LIN {X 0,Y 361.876,Z 72.401,A -85,B 0,C 180,E1 -13014.655,E2 -13014.655} C_VEL
LIN {X 0,Y 361.897,Z 72.531,A -85,B 0,C 180,E1 -13018.09,E2 -13018.09} C_VEL
LIN {X 0,Y 364.94,Z 85.338,A -85,B 0,C 180,E1 -13021.503,E2 -13021.503} C_VEL
LIN {X 0,Y 366.727,Z 94.642,A -85,B 0,C 180,E1 -13023.846,E2 -13023.846} C_VEL
LIN {X 0,Y 366.002,Z 102.488,A -85,B 0,C 180,E1 -13025.616,E2 -13025.616} C_VEL
LIN {X 0,Y 365.33,Z 108.755,A -85,B 0,C 180,E1 -13027.012,E2 -13027.012} C_VEL
LIN {X 0,Y 370.356,Z 135.443,A -85,B 0,C 180,E1 -13027.952,E2 -13027.952} C_VEL
LIN {X 0,Y 371.965,Z 146.662,A -85,B 0,C 180,E1 -13028.297,E2 -13028.297} C_VEL
LIN {X 0,Y 370.571,Z 218.065,A -85,B 0,C 180,E1 -13029.713,E2 -13029.713} C_VEL
LIN {X 0,Y 369.771,Z 231.878,A -85,B 0,C 180,E1 -13030.211,E2 -13030.211} C_VEL
LIN {X 0,Y 368.776,Z 244.274,A -85,B 0,C 180,E1 -13030.879,E2 -13030.879} C_VEL
LIN {X 0,Y 367.552,Z 256.145,A -85,B 0,C 180,E1 -13031.753,E2 -13031.753} C_VEL
LIN {X 0,Y 366.174,Z 267.553,A -85,B 0,C 180,E1 -13032.836,E2 -13032.836} C_VEL
LIN {X 0,Y 364.919,Z 277.858,A -85,B 0,C 180,E1 -13034.071,E2 -13034.071} C_VEL
LIN {X 0,Y 363.726,Z 287.134,A -85,B 0,C 180,E1 -13035.452,E2 -13035.452} C_VEL
LIN {X 0,Y 362.602,Z 296.152,A -85,B 0,C 180,E1 -13037.121,E2 -13037.121} C_VEL
LIN {X 0,Y 361.604,Z 303.436,A -85,B 0,C 180,E1 -13038.793,E2 -13038.793} C_VEL
LIN {X 0,Y 360.994,Z 309.293,A -85,B 0,C 180,E1 -13040.474,E2 -13040.474} C_VEL
LIN {X 0,Y 360.61,Z 313.923,A -85,B 0,C 180,E1 -13042.159,E2 -13042.159} C_VEL
LIN {X 0,Y 360.423,Z 317.693,A -85,B 0,C 180,E1 -13043.97,E2 -13043.97} C_VEL
LIN {X 0,Y 360.359,Z 320.002,A -85,B 0,C 180,E1 -13045.525,E2 -13045.525} C_VEL
LIN {X 0,Y 360.323,Z 321.192,A -85,B 0,C 180,E1 -13046.645,E2 -13046.645} C_VEL
LIN {X 0,Y 360.456,Z 322.312,A -85,B 0,C 180,E1 -13048.882,E2 -13048.882} C_VEL
LIN {X 0,Y 360.483,Z 322.289,A -85,B 0,C 180,E1 -13050,E2 -13050} C_VEL
LIN {X 0,Y 360.462,Z 321.871,A -85,B 0,C 180,E1 -13051.117,E2 -13051.117} C_VEL
LIN {X 0,Y 360.398,Z 321.01,A -85,B 0,C 180,E1 -13052.235,E2 -13052.235} C_VEL
LIN {X 0,Y 360.419,Z 318.073,A -85,B 0,C 180,E1 -13054.473,E2 -13054.473} C_VEL
LIN {X 0,Y 360.357,Z 314.691,A -85,B 0,C 180,E1 -13056.157,E2 -13056.157} C_VEL
LIN {X 0,Y 360.594,Z 310.228,A -85,B 0,C 180,E1 -13057.841,E2 -13057.841} C_VEL
LIN {X 0,Y 360.902,Z 304.546,A -85,B 0,C 180,E1 -13059.527,E2 -13059.527} C_VEL
LIN {X 0,Y 361.389,Z 297.422,A -85,B 0,C 180,E1 -13061.214,E2 -13061.214} C_VEL
LIN {X 0,Y 362.224,Z 288.522,A -85,B 0,C 180,E1 -13062.892,E2 -13062.892} C_VEL
LIN {X 0,Y 363.1,Z 279.397,A -85,B 0,C 180,E1 -13064.287,E2 -13064.287} C_VEL
LIN {X 0,Y 363.801,Z 269.428,A -85,B 0,C 180,E1 -13065.533,E2 -13065.533} C_VEL
LIN {X 0,Y 364.89,Z 258.101,A -85,B 0,C 180,E1 -13066.648,E2 -13066.648} C_VEL
LIN {X 0,Y 365.851,Z 245.515,A -85,B 0,C 180,E1 -13067.611,E2 -13067.611} C_VEL
LIN {X 0,Y 366.722,Z 232.662,A -85,B 0,C 180,E1 -13068.325,E2 -13068.325} C_VEL
LIN {X 0,Y 367.337,Z 218.902,A -85,B 0,C 180,E1 -13068.835,E2 -13068.835} C_VEL
LIN {X 0,Y 368.208,Z 162.822,A -85,B 0,C 180,E1 -13069.954,E2 -13069.954} C_VEL
LIN {X 0,Y 368.392,Z 143.971,A -85,B 0,C 180,E1 -13070.322,E2 -13070.322} C_VEL
LIN {X 0,Y 363.707,Z 109.248,A -85,B 0,C 180,E1 -13071.263,E2 -13071.263} C_VEL
LIN {X 0,Y 365.256,Z 90.835,A -85,B 0,C 180,E1 -13075.265,E2 -13075.265} C_VEL
LIN {X 0,Y 364.505,Z 85.088,A -85,B 0,C 180,E1 -13076.6,E2 -13076.6} C_VEL
LIN {X 0,Y 361.928,Z 72.512,A -85,B 0,C 180,E1 -13079.648,E2 -13079.648} C_VEL
LIN {X 0,Y 361.86,Z 72.408,A -85,B 0,C 180,E1 -13083.369,E2 -13083.369} C_VEL
LIN {X 0,Y 361.873,Z 72.406,A -85,B 0,C 180,E1 -13087.017,E2 -13087.017} C_VEL
LIN {X 0,Y 361.856,Z 72.412,A -85,B 0,C 180,E1 -13089.861,E2 -13089.861} C_VEL
LIN {X 0,Y 361.836,Z 72.41,A -85,B 0,C 180,E1 -13092.829,E2 -13092.829} C_VEL
LIN {X 0,Y 361.817,Z 72.414,A -85,B 0,C 180,E1 -13095.946,E2 -13095.946} C_VEL
LIN {X 0,Y 361.835,Z 72.415,A -85,B 0,C 180,E1 -13099.244,E2 -13099.244} C_VEL
LIN {X 0,Y 361.862,Z 72.408,A -85,B 0,C 180,E1 -13102.777,E2 -13102.777} C_VEL
LIN {X 0,Y 361.853,Z 72.409,A -85,B 0,C 180,E1 -13105.72,E2 -13105.72} C_VEL
LIN {X 0,Y 361.874,Z 72.406,A -85,B 0,C 180,E1 -13109.672,E2 -13109.672} C_VEL
LIN {X 0,Y 361.953,Z 72.397,A -85,B 0,C 180,E1 -13113.475,E2 -13113.475} C_VEL
LIN {X 0,Y 361.889,Z 72.406,A -85,B 0,C 180,E1 -13117.145,E2 -13117.145} C_VEL
LIN {X 0,Y 361.905,Z 72.407,A -85,B 0,C 180,E1 -13120.723,E2 -13120.723} C_VEL
LIN {X 0,Y 361.932,Z 72.4,A -85,B 0,C 180,E1 -13123.066,E2 -13123.066} C_VEL
LIN {X 0,Y 361.998,Z 72.396,A -85,B 0,C 180,E1 -13126.528,E2 -13126.528} C_VEL
LIN {X 0,Y 362.03,Z 72.387,A -85,B 0,C 180,E1 -13129.938,E2 -13129.938} C_VEL
LIN {X 0,Y 362.161,Z 72.369,A -85,B 0,C 180,E1 -13133.314,E2 -13133.314} C_VEL
LIN {X 0,Y 362.277,Z 72.357,A -85,B 0,C 180,E1 -13137.777,E2 -13137.777} C_VEL
LIN {X 0,Y 362.424,Z 72.342,A -85,B 0,C 180,E1 -13140,E2 -13140} C_VEL
LIN {X 0,Y 362.278,Z 72.359,A -85,B 0,C 180,E1 -13142.224,E2 -13142.224} C_VEL
LIN {X 0,Y 362.139,Z 72.372,A -85,B 0,C 180,E1 -13146.687,E2 -13146.687} C_VEL
LIN {X 0,Y 362,Z 72.393,A -85,B 0,C 180,E1 -13150.063,E2 -13150.063} C_VEL
LIN {X 0,Y 361.998,Z 72.393,A -85,B 0,C 180,E1 -13153.899,E2 -13153.899} C_VEL
LIN {X 0,Y 361.967,Z 72.396,A -85,B 0,C 180,E1 -13157.939,E2 -13157.939} C_VEL
LIN {X 0,Y 361.893,Z 72.406,A -85,B 0,C 180,E1 -13161.653,E2 -13161.653} C_VEL
LIN {X 0,Y 361.928,Z 72.405,A -85,B 0,C 180,E1 -13165.291,E2 -13165.291} C_VEL
LIN {X 0,Y 361.908,Z 72.402,A -85,B 0,C 180,E1 -13167.779,E2 -13167.779} C_VEL
LIN {X 0,Y 361.838,Z 72.411,A -85,B 0,C 180,E1 -13171.63,E2 -13171.63} C_VEL
LIN {X 0,Y 361.875,Z 72.408,A -85,B 0,C 180,E1 -13175.345,E2 -13175.345} C_VEL
LIN {X 0,Y 361.827,Z 72.415,A -85,B 0,C 180,E1 -13179.019,E2 -13179.019} C_VEL
LIN {X 0,Y 361.833,Z 72.415,A -85,B 0,C 180,E1 -13182.83,E2 -13182.83} C_VEL
LIN {X 0,Y 361.819,Z 72.413,A -85,B 0,C 180,E1 -13185.947,E2 -13185.947} C_VEL
LIN {X 0,Y 361.831,Z 72.411,A -85,B 0,C 180,E1 -13189.246,E2 -13189.246} C_VEL
LIN {X 0,Y 361.866,Z 72.407,A -85,B 0,C 180,E1 -13192.982,E2 -13192.982} C_VEL
LIN {X 0,Y 361.861,Z 72.41,A -85,B 0,C 180,E1 -13196.631,E2 -13196.631} C_VEL
LIN {X 0,Y 361.867,Z 72.407,A -85,B 0,C 180,E1 -13199.672,E2 -13199.672} C_VEL
LIN {X 0,Y 361.869,Z 72.407,A -85,B 0,C 180,E1 -13203.469,E2 -13203.469} C_VEL
LIN {X 0,Y 361.879,Z 72.405,A -85,B 0,C 180,E1 -13207.144,E2 -13207.144} C_VEL
LIN {X 0,Y 361.915,Z 72.4,A -85,B 0,C 180,E1 -13210.724,E2 -13210.724} C_VEL
LIN {X 0,Y 361.992,Z 72.529,A -85,B 0,C 180,E1 -13213.903,E2 -13213.903} C_VEL
LIN {X 0,Y 363.304,Z 79.279,A -85,B 0,C 180,E1 -13215.793,E2 -13215.793} C_VEL
LIN {X 0,Y 367.036,Z 91.537,A -85,B 0,C 180,E1 -13216.248,E2 -13216.248} C_VEL
LIN {X 0,Y 369.083,Z 102.968,A -85,B 0,C 180,E1 -13216.585,E2 -13216.585} C_VEL
LIN {X 0,Y 367.678,Z 186.211,A -85,B 0,C 180,E1 -13218.213,E2 -13218.213} C_VEL
LIN {X 0,Y 367.307,Z 199.331,A -85,B 0,C 180,E1 -13218.69,E2 -13218.69} C_VEL
LIN {X 0,Y 366.748,Z 210.843,A -85,B 0,C 180,E1 -13219.302,E2 -13219.302} C_VEL
LIN {X 0,Y 366.172,Z 221.465,A -85,B 0,C 180,E1 -13220.053,E2 -13220.053} C_VEL
LIN {X 0,Y 365.429,Z 232.147,A -85,B 0,C 180,E1 -13221.01,E2 -13221.01} C_VEL
LIN {X 0,Y 364.469,Z 243.07,A -85,B 0,C 180,E1 -13222.243,E2 -13222.243} C_VEL
LIN {X 0,Y 363.565,Z 252.825,A -85,B 0,C 180,E1 -13223.619,E2 -13223.619} C_VEL
LIN {X 0,Y 362.792,Z 260.826,A -85,B 0,C 180,E1 -13224.999,E2 -13224.999} C_VEL
LIN {X 0,Y 361.948,Z 268.696,A -85,B 0,C 180,E1 -13226.661,E2 -13226.661} C_VEL
LIN {X 0,Y 361.398,Z 274.977,A -85,B 0,C 180,E1 -13228.329,E2 -13228.329} C_VEL
LIN {X 0,Y 360.982,Z 279.978,A -85,B 0,C 180,E1 -13230,E2 -13230} C_VEL
LIN {X 0,Y 360.731,Z 283.862,A -85,B 0,C 180,E1 -13231.675,E2 -13231.675} C_VEL
LIN {X 0,Y 360.501,Z 286.736,A -85,B 0,C 180,E1 -13233.353,E2 -13233.353} C_VEL
LIN {X 0,Y 360.489,Z 288.092,A -85,B 0,C 180,E1 -13234.473,E2 -13234.473} C_VEL
LIN {X 0,Y 360.532,Z 289.417,A -85,B 0,C 180,E1 -13236.187,E2 -13236.187} C_VEL
LIN {X 0,Y 360.425,Z 289.835,A -85,B 0,C 180,E1 -13237.845,E2 -13237.845} C_VEL
LIN {X 0,Y 360.437,Z 289.599,A -85,B 0,C 180,E1 -13238.974,E2 -13238.974} C_VEL
LIN {X 0,Y 360.627,Z 287.966,A -85,B 0,C 180,E1 -13241.238,E2 -13241.238} C_VEL
LIN {X 0,Y 361.115,Z 284.969,A -85,B 0,C 180,E1 -13243.318,E2 -13243.318} C_VEL
LIN {X 0,Y 361.595,Z 280.929,A -85,B 0,C 180,E1 -13245.212,E2 -13245.212} C_VEL
LIN {X 0,Y 362.294,Z 276.088,A -85,B 0,C 180,E1 -13246.917,E2 -13246.917} C_VEL
LIN {X 0,Y 363.187,Z 269.564,A -85,B 0,C 180,E1 -13248.72,E2 -13248.72} C_VEL
LIN {X 0,Y 364.269,Z 261.912,A -85,B 0,C 180,E1 -13250.391,E2 -13250.391} C_VEL
LIN {X 0,Y 365.532,Z 252.545,A -85,B 0,C 180,E1 -13252.02,E2 -13252.02} C_VEL
LIN {X 0,Y 366.719,Z 242.183,A -85,B 0,C 180,E1 -13253.468,E2 -13253.468} C_VEL
LIN {X 0,Y 367.025,Z 240.037,A -85,B 0,C 180,E1 -13253.719,E2 -13253.719} C_VEL
LIN {X 0,Y 366.968,Z 235.366,A -85,B 0,C 180,E1 -13254.283,E2 -13254.283} C_VEL
LIN {X 0,Y 365.087,Z 227.638,A -85,B 0,C 180,E1 -13255.215,E2 -13255.215} C_VEL
LIN {X 0,Y 363.2,Z 219.555,A -85,B 0,C 180,E1 -13256.063,E2 -13256.063} C_VEL
LIN {X 0,Y 363.035,Z 214.302,A -85,B 0,C 180,E1 -13256.48,E2 -13256.48} C_VEL
LIN {X 0,Y 363.846,Z 202.088,A -85,B 0,C 180,E1 -13257.188,E2 -13257.188} C_VEL
LIN {X 0,Y 364.479,Z 189.545,A -85,B 0,C 180,E1 -13257.682,E2 -13257.682} C_VEL
LIN {X 0,Y 364.95,Z 169.01,A -85,B 0,C 180,E1 -13258.143,E2 -13258.143} C_VEL
LIN {X 0,Y 366.275,Z 106.198,A -85,B 0,C 180,E1 -13259.38,E2 -13259.38} C_VEL
LIN {X 0,Y 364.455,Z 99.45,A -85,B 0,C 180,E1 -13259.66,E2 -13259.66} C_VEL
LIN {X 0,Y 357.029,Z 81.913,A -85,B 0,C 180,E1 -13260.619,E2 -13260.619} C_VEL
LIN {X 0,Y 356.33,Z 80.075,A -85,B 0,C 180,E1 -13260.738,E2 -13260.738} C_VEL
LIN {X 0,Y 354.823,Z 73.287,A -85,B 0,C 180,E1 -13262.92,E2 -13262.92} C_VEL
LIN {X 0,Y 354.796,Z 73.291,A -85,B 0,C 180,E1 -13266.46,E2 -13266.46} C_VEL
LIN {X 0,Y 354.772,Z 73.295,A -85,B 0,C 180,E1 -13269.412,E2 -13269.412} C_VEL
LIN {X 0,Y 354.784,Z 73.291,A -85,B 0,C 180,E1 -13272.866,E2 -13272.866} C_VEL
LIN {X 0,Y 354.765,Z 73.289,A -85,B 0,C 180,E1 -13276.103,E2 -13276.103} C_VEL
LIN {X 0,Y 354.765,Z 73.291,A -85,B 0,C 180,E1 -13279.175,E2 -13279.175} C_VEL
LIN {X 0,Y 354.801,Z 73.288,A -85,B 0,C 180,E1 -13282.405,E2 -13282.405} C_VEL
LIN {X 0,Y 354.81,Z 73.283,A -85,B 0,C 180,E1 -13284.94,E2 -13284.94} C_VEL
LIN {X 0,Y 354.779,Z 73.284,A -85,B 0,C 180,E1 -13288.41,E2 -13288.41} C_VEL
LIN {X 0,Y 354.791,Z 73.286,A -85,B 0,C 180,E1 -13291.613,E2 -13291.613} C_VEL
LIN {X 0,Y 354.837,Z 73.282,A -85,B 0,C 180,E1 -13295.657,E2 -13295.657} C_VEL
LIN {X 0,Y 354.83,Z 73.287,A -85,B 0,C 180,E1 -13299.113,E2 -13299.113} C_VEL
LIN {X 0,Y 354.883,Z 73.27,A -85,B 0,C 180,E1 -13302.719,E2 -13302.719} C_VEL
LIN {X 0,Y 354.955,Z 73.27,A -85,B 0,C 180,E1 -13306.255,E2 -13306.255} C_VEL
LIN {X 0,Y 354.958,Z 73.265,A -85,B 0,C 180,E1 -13309.735,E2 -13309.735} C_VEL
LIN {X 0,Y 355.086,Z 73.243,A -85,B 0,C 180,E1 -13313.179,E2 -13313.179} C_VEL
LIN {X 0,Y 355.234,Z 73.235,A -85,B 0,C 180,E1 -13317.732,E2 -13317.732} C_VEL
LIN {X 0,Y 355.175,Z 73.236,A -85,B 0,C 180,E1 -13321.134,E2 -13321.134} C_VEL
LIN {X 0,Y 355.23,Z 73.238,A -85,B 0,C 180,E1 -13322.267,E2 -13322.267} C_VEL
LIN {X 0,Y 355.09,Z 73.245,A -85,B 0,C 180,E1 -13326.82,E2 -13326.82} C_VEL
LIN {X 0,Y 354.958,Z 73.263,A -85,B 0,C 180,E1 -13330.264,E2 -13330.264} C_VEL
LIN {X 0,Y 354.946,Z 73.271,A -85,B 0,C 180,E1 -13334.019,E2 -13334.019} C_VEL
LIN {X 0,Y 354.892,Z 73.273,A -85,B 0,C 180,E1 -13338.092,E2 -13338.092} C_VEL
LIN {X 0,Y 354.837,Z 73.274,A -85,B 0,C 180,E1 -13342.106,E2 -13342.106} C_VEL
LIN {X 0,Y 354.901,Z 73.272,A -85,B 0,C 180,E1 -13345.827,E2 -13345.827} C_VEL
LIN {X 0,Y 354.82,Z 73.285,A -85,B 0,C 180,E1 -13349.682,E2 -13349.682} C_VEL
LIN {X 0,Y 354.808,Z 73.285,A -85,B 0,C 180,E1 -13353.702,E2 -13353.702} C_VEL
LIN {X 0,Y 354.8,Z 73.267,A -85,B 0,C 180,E1 -13356.459,E2 -13356.459} C_VEL
LIN {X 0,Y 354.826,Z 73.286,A -85,B 0,C 180,E1 -13359.423,E2 -13359.423} C_VEL
LIN {X 0,Y 354.79,Z 73.292,A -85,B 0,C 180,E1 -13362.867,E2 -13362.867} C_VEL
LIN {X 0,Y 354.769,Z 73.29,A -85,B 0,C 180,E1 -13366.103,E2 -13366.103} C_VEL
LIN {X 0,Y 354.791,Z 73.288,A -85,B 0,C 180,E1 -13369.179,E2 -13369.179} C_VEL
LIN {X 0,Y 354.81,Z 73.286,A -85,B 0,C 180,E1 -13372.402,E2 -13372.402} C_VEL
LIN {X 0,Y 354.814,Z 73.282,A -85,B 0,C 180,E1 -13374.941,E2 -13374.941} C_VEL
LIN {X 0,Y 354.806,Z 73.307,A -85,B 0,C 180,E1 -13377.584,E2 -13377.584} C_VEL
LIN {X 0,Y 358.013,Z 86.717,A -85,B 0,C 180,E1 -13381.253,E2 -13381.253} C_VEL
LIN {X 0,Y 359.876,Z 96.303,A -85,B 0,C 180,E1 -13383.722,E2 -13383.722} C_VEL
LIN {X 0,Y 358.622,Z 108.094,A -85,B 0,C 180,E1 -13386.42,E2 -13386.42} C_VEL
LIN {X 0,Y 358.573,Z 108.532,A -85,B 0,C 180,E1 -13386.509,E2 -13386.509} C_VEL
LIN {X 0,Y 363.718,Z 135.365,A -85,B 0,C 180,E1 -13387.476,E2 -13387.476} C_VEL
LIN {X 0,Y 365.484,Z 147.486,A -85,B 0,C 180,E1 -13387.861,E2 -13387.861} C_VEL
LIN {X 0,Y 364.072,Z 217.142,A -85,B 0,C 180,E1 -13389.261,E2 -13389.261} C_VEL
LIN {X 0,Y 363.297,Z 230.396,A -85,B 0,C 180,E1 -13389.732,E2 -13389.732} C_VEL
LIN {X 0,Y 362.123,Z 243.672,A -85,B 0,C 180,E1 -13390.44,E2 -13390.44} C_VEL
LIN {X 0,Y 361.005,Z 254.823,A -85,B 0,C 180,E1 -13391.263,E2 -13391.263} C_VEL
LIN {X 0,Y 359.564,Z 266.413,A -85,B 0,C 180,E1 -13392.364,E2 -13392.364} C_VEL
LIN {X 0,Y 358.191,Z 276.856,A -85,B 0,C 180,E1 -13393.617,E2 -13393.617} C_VEL
LIN {X 0,Y 357.079,Z 285.167,A -85,B 0,C 180,E1 -13394.843,E2 -13394.843} C_VEL
LIN {X 0,Y 356.067,Z 293.317,A -85,B 0,C 180,E1 -13396.299,E2 -13396.299} C_VEL
LIN {X 0,Y 354.907,Z 301.072,A -85,B 0,C 180,E1 -13397.999,E2 -13397.999} C_VEL
LIN {X 0,Y 354.192,Z 307.312,A -85,B 0,C 180,E1 -13399.713,E2 -13399.713} C_VEL
LIN {X 0,Y 353.673,Z 312.291,A -85,B 0,C 180,E1 -13401.429,E2 -13401.429} C_VEL
LIN {X 0,Y 353.395,Z 316.155,A -85,B 0,C 180,E1 -13403.147,E2 -13403.147} C_VEL
LIN {X 0,Y 353.27,Z 319.745,A -85,B 0,C 180,E1 -13405.435,E2 -13405.435} C_VEL
LIN {X 0,Y 353.242,Z 320.908,A -85,B 0,C 180,E1 -13406.578,E2 -13406.578} C_VEL
LIN {X 0,Y 353.358,Z 321.998,A -85,B 0,C 180,E1 -13408.86,E2 -13408.86} C_VEL
LIN {X 0,Y 353.401,Z 321.962,A -85,B 0,C 180,E1 -13410,E2 -13410} C_VEL
LIN {X 0,Y 353.366,Z 321.52,A -85,B 0,C 180,E1 -13411.139,E2 -13411.139} C_VEL
LIN {X 0,Y 353.3,Z 320.639,A -85,B 0,C 180,E1 -13412.28,E2 -13412.28} C_VEL
LIN {X 0,Y 353.278,Z 319.359,A -85,B 0,C 180,E1 -13413.421,E2 -13413.421} C_VEL
LIN {X 0,Y 353.272,Z 316.635,A -85,B 0,C 180,E1 -13415.136,E2 -13415.136} C_VEL
LIN {X 0,Y 353.351,Z 312.875,A -85,B 0,C 180,E1 -13416.854,E2 -13416.854} C_VEL
LIN {X 0,Y 353.627,Z 307.982,A -85,B 0,C 180,E1 -13418.572,E2 -13418.572} C_VEL
LIN {X 0,Y 354.016,Z 301.801,A -85,B 0,C 180,E1 -13420.292,E2 -13420.292} C_VEL
LIN {X 0,Y 354.682,Z 294.114,A -85,B 0,C 180,E1 -13422.008,E2 -13422.008} C_VEL
LIN {X 0,Y 355.384,Z 286.236,A -85,B 0,C 180,E1 -13423.436,E2 -13423.436} C_VEL
LIN {X 0,Y 356.253,Z 276.602,A -85,B 0,C 180,E1 -13424.86,E2 -13424.86} C_VEL
LIN {X 0,Y 357.226,Z 265.914,A -85,B 0,C 180,E1 -13426.134,E2 -13426.134} C_VEL
LIN {X 0,Y 358.191,Z 255.609,A -85,B 0,C 180,E1 -13427.116,E2 -13427.116} C_VEL
LIN {X 0,Y 359.138,Z 243.357,A -85,B 0,C 180,E1 -13428.025,E2 -13428.025} C_VEL
LIN {X 0,Y 360.052,Z 230.478,A -85,B 0,C 180,E1 -13428.714,E2 -13428.714} C_VEL
LIN {X 0,Y 360.57,Z 216.855,A -85,B 0,C 180,E1 -13429.203,E2 -13429.203} C_VEL
LIN {X 0,Y 361.606,Z 144.583,A -85,B 0,C 180,E1 -13430.648,E2 -13430.648} C_VEL
LIN {X 0,Y 356.785,Z 108.9,A -85,B 0,C 180,E1 -13431.645,E2 -13431.645} C_VEL
LIN {X 0,Y 358.294,Z 92.067,A -85,B 0,C 180,E1 -13435.375,E2 -13435.375} C_VEL
LIN {X 0,Y 357.421,Z 85.709,A -85,B 0,C 180,E1 -13436.888,E2 -13436.888} C_VEL
LIN {X 0,Y 354.849,Z 73.318,A -85,B 0,C 180,E1 -13439.965,E2 -13439.965} C_VEL
LIN {X 0,Y 354.806,Z 73.29,A -85,B 0,C 180,E1 -13443.702,E2 -13443.702} C_VEL
LIN {X 0,Y 354.801,Z 73.287,A -85,B 0,C 180,E1 -13446.459,E2 -13446.459} C_VEL
LIN {X 0,Y 354.823,Z 73.287,A -85,B 0,C 180,E1 -13449.423,E2 -13449.423} C_VEL
LIN {X 0,Y 354.788,Z 73.288,A -85,B 0,C 180,E1 -13452.867,E2 -13452.867} C_VEL
LIN {X 0,Y 354.766,Z 73.291,A -85,B 0,C 180,E1 -13456.103,E2 -13456.103} C_VEL
LIN {X 0,Y 354.787,Z 73.292,A -85,B 0,C 180,E1 -13459.179,E2 -13459.179} C_VEL
LIN {X 0,Y 354.806,Z 73.286,A -85,B 0,C 180,E1 -13462.402,E2 -13462.402} C_VEL
LIN {X 0,Y 354.811,Z 73.288,A -85,B 0,C 180,E1 -13464.941,E2 -13464.941} C_VEL
LIN {X 0,Y 354.792,Z 73.288,A -85,B 0,C 180,E1 -13468.405,E2 -13468.405} C_VEL
LIN {X 0,Y 354.848,Z 73.281,A -85,B 0,C 180,E1 -13471.619,E2 -13471.619} C_VEL
LIN {X 0,Y 354.898,Z 73.274,A -85,B 0,C 180,E1 -13474.173,E2 -13474.173} C_VEL
LIN {X 0,Y 354.834,Z 73.282,A -85,B 0,C 180,E1 -13477.894,E2 -13477.894} C_VEL
LIN {X 0,Y 354.921,Z 73.271,A -85,B 0,C 180,E1 -13481.892,E2 -13481.892} C_VEL
LIN {X 0,Y 354.942,Z 73.27,A -85,B 0,C 180,E1 -13485.981,E2 -13485.981} C_VEL
LIN {X 0,Y 354.977,Z 73.265,A -85,B 0,C 180,E1 -13489.736,E2 -13489.736} C_VEL
LIN {X 0,Y 355.124,Z 73.246,A -85,B 0,C 180,E1 -13493.181,E2 -13493.181} C_VEL
LIN {X 0,Y 355.24,Z 73.233,A -85,B 0,C 180,E1 -13497.733,E2 -13497.733} C_VEL
LIN {X 0,Y 355.373,Z 73.22,A -85,B 0,C 180,E1 -13500,E2 -13500} C_VEL
LIN {X 0,Y 355.241,Z 73.235,A -85,B 0,C 180,E1 -13502.268,E2 -13502.268} C_VEL
LIN {X 0,Y 355.103,Z 73.249,A -85,B 0,C 180,E1 -13506.82,E2 -13506.82} C_VEL
LIN {X 0,Y 354.956,Z 73.268,A -85,B 0,C 180,E1 -13510.265,E2 -13510.265} C_VEL
LIN {X 0,Y 354.943,Z 73.271,A -85,B 0,C 180,E1 -13514.019,E2 -13514.019} C_VEL
LIN {X 0,Y 354.922,Z 73.272,A -85,B 0,C 180,E1 -13518.109,E2 -13518.109} C_VEL
LIN {X 0,Y 354.836,Z 73.282,A -85,B 0,C 180,E1 -13522.106,E2 -13522.106} C_VEL
LIN {X 0,Y 354.899,Z 73.275,A -85,B 0,C 180,E1 -13525.828,E2 -13525.828} C_VEL
LIN {X 0,Y 354.818,Z 73.285,A -85,B 0,C 180,E1 -13529.682,E2 -13529.682} C_VEL
LIN {X 0,Y 354.807,Z 73.286,A -85,B 0,C 180,E1 -13533.702,E2 -13533.702} C_VEL
LIN {X 0,Y 354.797,Z 73.288,A -85,B 0,C 180,E1 -13536.46,E2 -13536.46} C_VEL
LIN {X 0,Y 354.768,Z 73.291,A -85,B 0,C 180,E1 -13539.413,E2 -13539.413} C_VEL
LIN {X 0,Y 354.786,Z 73.293,A -85,B 0,C 180,E1 -13542.867,E2 -13542.867} C_VEL
LIN {X 0,Y 354.768,Z 73.292,A -85,B 0,C 180,E1 -13546.104,E2 -13546.104} C_VEL
LIN {X 0,Y 354.783,Z 73.289,A -85,B 0,C 180,E1 -13549.179,E2 -13549.179} C_VEL
LIN {X 0,Y 354.803,Z 73.292,A -85,B 0,C 180,E1 -13552.404,E2 -13552.404} C_VEL
LIN {X 0,Y 354.814,Z 73.286,A -85,B 0,C 180,E1 -13554.941,E2 -13554.941} C_VEL
LIN {X 0,Y 354.796,Z 73.291,A -85,B 0,C 180,E1 -13558.406,E2 -13558.406} C_VEL
LIN {X 0,Y 354.804,Z 73.287,A -85,B 0,C 180,E1 -13561.615,E2 -13561.615} C_VEL
LIN {X 0,Y 354.808,Z 73.286,A -85,B 0,C 180,E1 -13565.42,E2 -13565.42} C_VEL
LIN {X 0,Y 354.83,Z 73.283,A -85,B 0,C 180,E1 -13569.114,E2 -13569.114} C_VEL
LIN {X 0,Y 354.902,Z 73.28,A -85,B 0,C 180,E1 -13572.72,E2 -13572.72} C_VEL
LIN {X 0,Y 354.933,Z 73.314,A -85,B 0,C 180,E1 -13573.611,E2 -13573.611} C_VEL
LIN {X 0,Y 356.127,Z 79.587,A -85,B 0,C 180,E1 -13575.4,E2 -13575.4} C_VEL
LIN {X 0,Y 360.444,Z 93.244,A -85,B 0,C 180,E1 -13575.932,E2 -13575.932} C_VEL
LIN {X 0,Y 362.291,Z 102.702,A -85,B 0,C 180,E1 -13576.226,E2 -13576.226} C_VEL
LIN {X 0,Y 360.875,Z 187.104,A -85,B 0,C 180,E1 -13577.916,E2 -13577.916} C_VEL
LIN {X 0,Y 360.41,Z 200.803,A -85,B 0,C 180,E1 -13578.435,E2 -13578.435} C_VEL
LIN {X 0,Y 359.86,Z 212.564,A -85,B 0,C 180,E1 -13579.095,E2 -13579.095} C_VEL
LIN {X 0,Y 359.197,Z 224.493,A -85,B 0,C 180,E1 -13580,E2 -13580} C_VEL
LIN {X 0,Y 358.264,Z 235.895,A -85,B 0,C 180,E1 -13581.114,E2 -13581.114} C_VEL
LIN {X 0,Y 357.326,Z 246.172,A -85,B 0,C 180,E1 -13582.371,E2 -13582.371} C_VEL
LIN {X 0,Y 356.383,Z 255.426,A -85,B 0,C 180,E1 -13583.774,E2 -13583.774} C_VEL
LIN {X 0,Y 355.408,Z 264.378,A -85,B 0,C 180,E1 -13585.464,E2 -13585.464} C_VEL
LIN {X 0,Y 354.705,Z 271.592,A -85,B 0,C 180,E1 -13587.161,E2 -13587.161} C_VEL
LIN {X 0,Y 354.143,Z 277.377,A -85,B 0,C 180,E1 -13588.863,E2 -13588.863} C_VEL
LIN {X 0,Y 353.81,Z 281.933,A -85,B 0,C 180,E1 -13590.569,E2 -13590.569} C_VEL
LIN {X 0,Y 353.592,Z 285.408,A -85,B 0,C 180,E1 -13592.279,E2 -13592.279} C_VEL
LIN {X 0,Y 353.41,Z 287.171,A -85,B 0,C 180,E1 -13593.421,E2 -13593.421} C_VEL
LIN {X 0,Y 353.417,Z 288.501,A -85,B 0,C 180,E1 -13594.563,E2 -13594.563} C_VEL
LIN {X 0,Y 353.452,Z 289.716,A -85,B 0,C 180,E1 -13596.171,E2 -13596.171} C_VEL
LIN {X 0,Y 353.332,Z 290.145,A -85,B 0,C 180,E1 -13598.004,E2 -13598.004} C_VEL
LIN {X 0,Y 353.357,Z 289.883,A -85,B 0,C 180,E1 -13599.156,E2 -13599.156} C_VEL
LIN {X 0,Y 353.583,Z 288.197,A -85,B 0,C 180,E1 -13601.465,E2 -13601.465} C_VEL
LIN {X 0,Y 354.055,Z 285.414,A -85,B 0,C 180,E1 -13603.428,E2 -13603.428} C_VEL
LIN {X 0,Y 354.632,Z 281.025,A -85,B 0,C 180,E1 -13605.518,E2 -13605.518} C_VEL
LIN {X 0,Y 355.394,Z 276.123,A -85,B 0,C 180,E1 -13607.256,E2 -13607.256} C_VEL
LIN {X 0,Y 356.286,Z 269.812,A -85,B 0,C 180,E1 -13609.022,E2 -13609.022} C_VEL
LIN {X 0,Y 357.474,Z 262.121,A -85,B 0,C 180,E1 -13610.725,E2 -13610.725} C_VEL
LIN {X 0,Y 358.604,Z 254.102,A -85,B 0,C 180,E1 -13612.165,E2 -13612.165} C_VEL
LIN {X 0,Y 359.894,Z 243.469,A -85,B 0,C 180,E1 -13613.712,E2 -13613.712} C_VEL
LIN {X 0,Y 361.133,Z 233.264,A -85,B 0,C 180,E1 -13614.888,E2 -13614.888} C_VEL
LIN {X 0,Y 362.267,Z 222.413,A -85,B 0,C 180,E1 -13615.881,E2 -13615.881} C_VEL
LIN {X 0,Y 363.035,Z 214.302,A -85,B 0,C 180,E1 -13616.48,E2 -13616.48} C_VEL
LIN {X 0,Y 362.72,Z 210.721,A -85,B 0,C 180,E1 -13616.757,E2 -13616.757} C_VEL
LIN {X 0,Y 360.441,Z 205.186,A -85,B 0,C 180,E1 -13617.264,E2 -13617.264} C_VEL
LIN {X 0,Y 358.124,Z 199.528,A -85,B 0,C 180,E1 -13617.723,E2 -13617.723} C_VEL
LIN {X 0,Y 357.729,Z 195.765,A -85,B 0,C 180,E1 -13617.919,E2 -13617.919} C_VEL
LIN {X 0,Y 358.26,Z 182.186,A -85,B 0,C 180,E1 -13618.334,E2 -13618.334} C_VEL
LIN {X 0,Y 359.803,Z 107.144,A -85,B 0,C 180,E1 -13619.848,E2 -13619.848} C_VEL
LIN {X 0,Y 357.965,Z 101.016,A -85,B 0,C 180,E1 -13620.124,E2 -13620.124} C_VEL
LIN {X 0,Y 350.366,Z 83.313,A -85,B 0,C 180,E1 -13621.134,E2 -13621.134} C_VEL
LIN {X 0,Y 349.147,Z 80.374,A -85,B 0,C 180,E1 -13621.339,E2 -13621.339} C_VEL
LIN {X 0,Y 347.768,Z 74.17,A -85,B 0,C 180,E1 -13623.353,E2 -13623.353} C_VEL
LIN {X 0,Y 347.769,Z 74.171,A -85,B 0,C 180,E1 -13626.064,E2 -13626.064} C_VEL
LIN {X 0,Y 347.734,Z 74.171,A -85,B 0,C 180,E1 -13628.796,E2 -13628.796} C_VEL
LIN {X 0,Y 347.743,Z 74.169,A -85,B 0,C 180,E1 -13631.832,E2 -13631.832} C_VEL
LIN {X 0,Y 347.702,Z 74.158,A -85,B 0,C 180,E1 -13635.028,E2 -13635.028} C_VEL
LIN {X 0,Y 347.741,Z 74.164,A -85,B 0,C 180,E1 -13638.4,E2 -13638.4} C_VEL
LIN {X 0,Y 347.764,Z 74.165,A -85,B 0,C 180,E1 -13642.014,E2 -13642.014} C_VEL
LIN {X 0,Y 347.746,Z 74.167,A -85,B 0,C 180,E1 -13645.536,E2 -13645.536} C_VEL
LIN {X 0,Y 347.733,Z 74.162,A -85,B 0,C 180,E1 -13648.299,E2 -13648.299} C_VEL
LIN {X 0,Y 347.744,Z 74.171,A -85,B 0,C 180,E1 -13650.984,E2 -13650.984} C_VEL
LIN {X 0,Y 347.769,Z 74.167,A -85,B 0,C 180,E1 -13654.888,E2 -13654.888} C_VEL
LIN {X 0,Y 347.782,Z 74.159,A -85,B 0,C 180,E1 -13658.669,E2 -13658.669} C_VEL
LIN {X 0,Y 347.846,Z 74.146,A -85,B 0,C 180,E1 -13662.358,E2 -13662.358} C_VEL
LIN {X 0,Y 347.901,Z 74.147,A -85,B 0,C 180,E1 -13665.971,E2 -13665.971} C_VEL
LIN {X 0,Y 347.899,Z 74.145,A -85,B 0,C 180,E1 -13669.524,E2 -13669.524} C_VEL
LIN {X 0,Y 348.053,Z 74.119,A -85,B 0,C 180,E1 -13673.041,E2 -13673.041} C_VEL
LIN {X 0,Y 348.196,Z 74.111,A -85,B 0,C 180,E1 -13677.686,E2 -13677.686} C_VEL
LIN {X 0,Y 348.143,Z 74.112,A -85,B 0,C 180,E1 -13681.156,E2 -13681.156} C_VEL
LIN {X 0,Y 348.191,Z 74.115,A -85,B 0,C 180,E1 -13682.313,E2 -13682.313} C_VEL
LIN {X 0,Y 348.057,Z 74.121,A -85,B 0,C 180,E1 -13686.958,E2 -13686.958} C_VEL
LIN {X 0,Y 347.899,Z 74.141,A -85,B 0,C 180,E1 -13690.475,E2 -13690.475} C_VEL
LIN {X 0,Y 347.902,Z 74.147,A -85,B 0,C 180,E1 -13694.15,E2 -13694.15} C_VEL
LIN {X 0,Y 347.832,Z 74.153,A -85,B 0,C 180,E1 -13698.259,E2 -13698.259} C_VEL
LIN {X 0,Y 347.791,Z 74.154,A -85,B 0,C 180,E1 -13701.635,E2 -13701.635} C_VEL
LIN {X 0,Y 347.815,Z 74.162,A -85,B 0,C 180,E1 -13705.108,E2 -13705.108} C_VEL
LIN {X 0,Y 347.811,Z 74.158,A -85,B 0,C 180,E1 -13707.694,E2 -13707.694} C_VEL
LIN {X 0,Y 347.752,Z 74.164,A -85,B 0,C 180,E1 -13710.348,E2 -13710.348} C_VEL
LIN {X 0,Y 347.75,Z 74.164,A -85,B 0,C 180,E1 -13714.044,E2 -13714.044} C_VEL
LIN {X 0,Y 347.764,Z 74.147,A -85,B 0,C 180,E1 -13717.321,E2 -13717.321} C_VEL
LIN {X 0,Y 347.735,Z 74.171,A -85,B 0,C 180,E1 -13720.297,E2 -13720.297} C_VEL
LIN {X 0,Y 347.725,Z 74.17,A -85,B 0,C 180,E1 -13723.408,E2 -13723.408} C_VEL
LIN {X 0,Y 347.727,Z 74.168,A -85,B 0,C 180,E1 -13726.686,E2 -13726.686} C_VEL
LIN {X 0,Y 347.75,Z 74.164,A -85,B 0,C 180,E1 -13730.173,E2 -13730.173} C_VEL
LIN {X 0,Y 347.764,Z 74.165,A -85,B 0,C 180,E1 -13732.679,E2 -13732.679} C_VEL
LIN {X 0,Y 347.75,Z 74.172,A -85,B 0,C 180,E1 -13735.956,E2 -13735.956} C_VEL
LIN {X 0,Y 347.789,Z 74.256,A -85,B 0,C 180,E1 -13737.11,E2 -13737.11} C_VEL
LIN {X 0,Y 350.777,Z 86.652,A -85,B 0,C 180,E1 -13740.602,E2 -13740.602} C_VEL
LIN {X 0,Y 352.847,Z 96.905,A -85,B 0,C 180,E1 -13743.322,E2 -13743.322} C_VEL
LIN {X 0,Y 352.904,Z 99.733,A -85,B 0,C 180,E1 -13744.015,E2 -13744.015} C_VEL
LIN {X 0,Y 351.88,Z 108.223,A -85,B 0,C 180,E1 -13745.973,E2 -13745.973} C_VEL
LIN {X 0,Y 357.333,Z 136.688,A -85,B 0,C 180,E1 -13747.029,E2 -13747.029} C_VEL
LIN {X 0,Y 359.019,Z 148.271,A -85,B 0,C 180,E1 -13747.408,E2 -13747.408} C_VEL
LIN {X 0,Y 357.527,Z 217.38,A -85,B 0,C 180,E1 -13748.826,E2 -13748.826} C_VEL
LIN {X 0,Y 356.731,Z 230.444,A -85,B 0,C 180,E1 -13749.305,E2 -13749.305} C_VEL
LIN {X 0,Y 355.591,Z 243.061,A -85,B 0,C 180,E1 -13749.991,E2 -13749.991} C_VEL
LIN {X 0,Y 354.312,Z 255.085,A -85,B 0,C 180,E1 -13750.895,E2 -13750.895} C_VEL
LIN {X 0,Y 352.816,Z 266.566,A -85,B 0,C 180,E1 -13752.015,E2 -13752.015} C_VEL
LIN {X 0,Y 351.364,Z 276.927,A -85,B 0,C 180,E1 -13753.289,E2 -13753.289} C_VEL
LIN {X 0,Y 350.136,Z 285.791,A -85,B 0,C 180,E1 -13754.64,E2 -13754.64} C_VEL
LIN {X 0,Y 348.96,Z 294.642,A -85,B 0,C 180,E1 -13756.311,E2 -13756.311} C_VEL
LIN {X 0,Y 347.781,Z 302.075,A -85,B 0,C 180,E1 -13758.045,E2 -13758.045} C_VEL
LIN {X 0,Y 346.961,Z 308.958,A -85,B 0,C 180,E1 -13760.085,E2 -13760.085} C_VEL
LIN {X 0,Y 346.497,Z 313.517,A -85,B 0,C 180,E1 -13761.837,E2 -13761.837} C_VEL
LIN {X 0,Y 346.234,Z 317.73,A -85,B 0,C 180,E1 -13764.056,E2 -13764.056} C_VEL
LIN {X 0,Y 346.167,Z 319.487,A -85,B 0,C 180,E1 -13765.342,E2 -13765.342} C_VEL
LIN {X 0,Y 346.163,Z 320.623,A -85,B 0,C 180,E1 -13766.508,E2 -13766.508} C_VEL
LIN {X 0,Y 346.26,Z 321.684,A -85,B 0,C 180,E1 -13768.837,E2 -13768.837} C_VEL
LIN {X 0,Y 346.322,Z 321.635,A -85,B 0,C 180,E1 -13770,E2 -13770} C_VEL
LIN {X 0,Y 346.27,Z 321.165,A -85,B 0,C 180,E1 -13771.163,E2 -13771.163} C_VEL
LIN {X 0,Y 346.199,Z 318.974,A -85,B 0,C 180,E1 -13773.491,E2 -13773.491} C_VEL
LIN {X 0,Y 346.155,Z 315.869,A -85,B 0,C 180,E1 -13775.429,E2 -13775.429} C_VEL
LIN {X 0,Y 346.37,Z 310.928,A -85,B 0,C 180,E1 -13777.578,E2 -13777.578} C_VEL
LIN {X 0,Y 346.743,Z 304.558,A -85,B 0,C 180,E1 -13779.626,E2 -13779.626} C_VEL
LIN {X 0,Y 347.252,Z 297.614,A -85,B 0,C 180,E1 -13781.38,E2 -13781.38} C_VEL
LIN {X 0,Y 348.012,Z 290.531,A -85,B 0,C 180,E1 -13782.835,E2 -13782.835} C_VEL
LIN {X 0,Y 348.837,Z 282.36,A -85,B 0,C 180,E1 -13784.227,E2 -13784.227} C_VEL
LIN {X 0,Y 349.648,Z 272.567,A -85,B 0,C 180,E1 -13785.595,E2 -13785.595} C_VEL
LIN {X 0,Y 350.636,Z 262.342,A -85,B 0,C 180,E1 -13786.745,E2 -13786.745} C_VEL
LIN {X 0,Y 351.68,Z 251.187,A -85,B 0,C 180,E1 -13787.743,E2 -13787.743} C_VEL
LIN {X 0,Y 352.606,Z 238.772,A -85,B 0,C 180,E1 -13788.596,E2 -13788.596} C_VEL
LIN {X 0,Y 353.464,Z 225.581,A -85,B 0,C 180,E1 -13789.227,E2 -13789.227} C_VEL
LIN {X 0,Y 353.865,Z 212.807,A -85,B 0,C 180,E1 -13789.619,E2 -13789.619} C_VEL
LIN {X 0,Y 354.856,Z 145.344,A -85,B 0,C 180,E1 -13790.98,E2 -13790.98} C_VEL
LIN {X 0,Y 350.018,Z 109.751,A -85,B 0,C 180,E1 -13791.994,E2 -13791.994} C_VEL
LIN {X 0,Y 349.858,Z 108.546,A -85,B 0,C 180,E1 -13792.042,E2 -13792.042} C_VEL
LIN {X 0,Y 351.273,Z 93.78,A -85,B 0,C 180,E1 -13795.381,E2 -13795.381} C_VEL
LIN {X 0,Y 351.121,Z 90.627,A -85,B 0,C 180,E1 -13796.126,E2 -13796.126} C_VEL
LIN {X 0,Y 348.607,Z 77.794,A -85,B 0,C 180,E1 -13799.34,E2 -13799.34} C_VEL
LIN {X 0,Y 347.817,Z 74.162,A -85,B 0,C 180,E1 -13800.297,E2 -13800.297} C_VEL
LIN {X 0,Y 347.744,Z 74.167,A -85,B 0,C 180,E1 -13804.464,E2 -13804.464} C_VEL
LIN {X 0,Y 347.777,Z 74.165,A -85,B 0,C 180,E1 -13807.989,E2 -13807.989} C_VEL
LIN {X 0,Y 347.75,Z 74.168,A -85,B 0,C 180,E1 -13811.83,E2 -13811.83} C_VEL
LIN {X 0,Y 347.705,Z 74.172,A -85,B 0,C 180,E1 -13815.027,E2 -13815.027} C_VEL
LIN {X 0,Y 347.749,Z 74.165,A -85,B 0,C 180,E1 -13818.397,E2 -13818.397} C_VEL
LIN {X 0,Y 347.772,Z 74.162,A -85,B 0,C 180,E1 -13822.011,E2 -13822.011} C_VEL
LIN {X 0,Y 347.743,Z 74.168,A -85,B 0,C 180,E1 -13825.536,E2 -13825.536} C_VEL
LIN {X 0,Y 347.763,Z 74.164,A -85,B 0,C 180,E1 -13829.654,E2 -13829.654} C_VEL
LIN {X 0,Y 347.85,Z 74.156,A -85,B 0,C 180,E1 -13832.745,E2 -13832.745} C_VEL
LIN {X 0,Y 347.788,Z 74.16,A -85,B 0,C 180,E1 -13836.162,E2 -13836.162} C_VEL
LIN {X 0,Y 347.811,Z 74.157,A -85,B 0,C 180,E1 -13839.909,E2 -13839.909} C_VEL
LIN {X 0,Y 347.865,Z 74.153,A -85,B 0,C 180,E1 -13842.359,E2 -13842.359} C_VEL
LIN {X 0,Y 347.896,Z 74.147,A -85,B 0,C 180,E1 -13845.971,E2 -13845.971} C_VEL
LIN {X 0,Y 347.928,Z 74.142,A -85,B 0,C 180,E1 -13849.526,E2 -13849.526} C_VEL
LIN {X 0,Y 348.09,Z 74.123,A -85,B 0,C 180,E1 -13853.042,E2 -13853.042} C_VEL
LIN {X 0,Y 348.203,Z 74.11,A -85,B 0,C 180,E1 -13857.687,E2 -13857.687} C_VEL
LIN {X 0,Y 348.323,Z 74.098,A -85,B 0,C 180,E1 -13860,E2 -13860} C_VEL
LIN {X 0,Y 348.203,Z 74.111,A -85,B 0,C 180,E1 -13862.314,E2 -13862.314} C_VEL
LIN {X 0,Y 348.07,Z 74.125,A -85,B 0,C 180,E1 -13866.959,E2 -13866.959} C_VEL
LIN {X 0,Y 347.896,Z 74.147,A -85,B 0,C 180,E1 -13870.476,E2 -13870.476} C_VEL
LIN {X 0,Y 347.898,Z 74.147,A -85,B 0,C 180,E1 -13874.15,E2 -13874.15} C_VEL
LIN {X 0,Y 347.891,Z 74.147,A -85,B 0,C 180,E1 -13878.29,E2 -13878.29} C_VEL
LIN {X 0,Y 347.79,Z 74.163,A -85,B 0,C 180,E1 -13881.636,E2 -13881.636} C_VEL
LIN {X 0,Y 347.812,Z 74.161,A -85,B 0,C 180,E1 -13885.109,E2 -13885.109} C_VEL
LIN {X 0,Y 347.808,Z 74.159,A -85,B 0,C 180,E1 -13887.695,E2 -13887.695} C_VEL
LIN {X 0,Y 347.75,Z 74.165,A -85,B 0,C 180,E1 -13890.348,E2 -13890.348} C_VEL
LIN {X 0,Y 347.749,Z 74.165,A -85,B 0,C 180,E1 -13894.044,E2 -13894.044} C_VEL
LIN {X 0,Y 347.757,Z 74.166,A -85,B 0,C 180,E1 -13897.322,E2 -13897.322} C_VEL
LIN {X 0,Y 347.742,Z 74.166,A -85,B 0,C 180,E1 -13901.602,E2 -13901.602} C_VEL
LIN {X 0,Y 347.706,Z 74.173,A -85,B 0,C 180,E1 -13905.027,E2 -13905.027} C_VEL
LIN {X 0,Y 347.748,Z 74.169,A -85,B 0,C 180,E1 -13908.398,E2 -13908.398} C_VEL
LIN {X 0,Y 347.765,Z 74.165,A -85,B 0,C 180,E1 -13912.014,E2 -13912.014} C_VEL
LIN {X 0,Y 347.746,Z 74.165,A -85,B 0,C 180,E1 -13915.537,E2 -13915.537} C_VEL
LIN {X 0,Y 347.747,Z 74.17,A -85,B 0,C 180,E1 -13918.301,E2 -13918.301} C_VEL
LIN {X 0,Y 347.748,Z 74.164,A -85,B 0,C 180,E1 -13920.985,E2 -13920.985} C_VEL
LIN {X 0,Y 347.749,Z 74.166,A -85,B 0,C 180,E1 -13923.601,E2 -13923.601} C_VEL
LIN {X 0,Y 347.755,Z 74.169,A -85,B 0,C 180,E1 -13926.16,E2 -13926.16} C_VEL
LIN {X 0,Y 347.812,Z 74.163,A -85,B 0,C 180,E1 -13929.91,E2 -13929.91} C_VEL
LIN {X 0,Y 347.871,Z 74.155,A -85,B 0,C 180,E1 -13932.966,E2 -13932.966} C_VEL
LIN {X 0,Y 347.863,Z 74.234,A -85,B 0,C 180,E1 -13933.344,E2 -13933.344} C_VEL
LIN {X 0,Y 349.01,Z 79.865,A -85,B 0,C 180,E1 -13934.987,E2 -13934.987} C_VEL
LIN {X 0,Y 353.881,Z 94.986,A -85,B 0,C 180,E1 -13935.607,E2 -13935.607} C_VEL
LIN {X 0,Y 355.599,Z 104.353,A -85,B 0,C 180,E1 -13935.899,E2 -13935.899} C_VEL
LIN {X 0,Y 354.124,Z 186.849,A -85,B 0,C 180,E1 -13937.573,E2 -13937.573} C_VEL
LIN {X 0,Y 353.743,Z 199.218,A -85,B 0,C 180,E1 -13938.032,E2 -13938.032} C_VEL
LIN {X 0,Y 353.076,Z 212.044,A -85,B 0,C 180,E1 -13938.737,E2 -13938.737} C_VEL
LIN {X 0,Y 352.354,Z 224.229,A -85,B 0,C 180,E1 -13939.659,E2 -13939.659} C_VEL
LIN {X 0,Y 351.394,Z 235.737,A -85,B 0,C 180,E1 -13940.793,E2 -13940.793} C_VEL
LIN {X 0,Y 350.427,Z 246.095,A -85,B 0,C 180,E1 -13942.075,E2 -13942.075} C_VEL
LIN {X 0,Y 349.551,Z 254.572,A -85,B 0,C 180,E1 -13943.362,E2 -13943.362} C_VEL
LIN {X 0,Y 348.74,Z 262.389,A -85,B 0,C 180,E1 -13944.797,E2 -13944.797} C_VEL
LIN {X 0,Y 347.837,Z 270.047,A -85,B 0,C 180,E1 -13946.525,E2 -13946.525} C_VEL
LIN {X 0,Y 347.244,Z 276.182,A -85,B 0,C 180,E1 -13948.261,E2 -13948.261} C_VEL
LIN {X 0,Y 346.805,Z 281.064,A -85,B 0,C 180,E1 -13950,E2 -13950} C_VEL
LIN {X 0,Y 346.572,Z 284.834,A -85,B 0,C 180,E1 -13951.743,E2 -13951.743} C_VEL
LIN {X 0,Y 346.323,Z 287.605,A -85,B 0,C 180,E1 -13953.491,E2 -13953.491} C_VEL
LIN {X 0,Y 346.325,Z 288.91,A -85,B 0,C 180,E1 -13954.656,E2 -13954.656} C_VEL
LIN {X 0,Y 346.372,Z 290.015,A -85,B 0,C 180,E1 -13956.155,E2 -13956.155} C_VEL
LIN {X 0,Y 346.259,Z 290.454,A -85,B 0,C 180,E1 -13958.169,E2 -13958.169} C_VEL
LIN {X 0,Y 346.336,Z 289.498,A -85,B 0,C 180,E1 -13960.523,E2 -13960.523} C_VEL
LIN {X 0,Y 346.553,Z 288.415,A -85,B 0,C 180,E1 -13961.701,E2 -13961.701} C_VEL
LIN {X 0,Y 347.022,Z 285.826,A -85,B 0,C 180,E1 -13963.561,E2 -13963.561} C_VEL
LIN {X 0,Y 347.459,Z 282.54,A -85,B 0,C 180,E1 -13965.245,E2 -13965.245} C_VEL
LIN {X 0,Y 348.212,Z 277.974,A -85,B 0,C 180,E1 -13967.017,E2 -13967.017} C_VEL
LIN {X 0,Y 349.165,Z 271.677,A -85,B 0,C 180,E1 -13968.91,E2 -13968.91} C_VEL
LIN {X 0,Y 350.222,Z 264.796,A -85,B 0,C 180,E1 -13970.56,E2 -13970.56} C_VEL
LIN {X 0,Y 351.647,Z 255.647,A -85,B 0,C 180,E1 -13972.318,E2 -13972.318} C_VEL
LIN {X 0,Y 352.922,Z 246.086,A -85,B 0,C 180,E1 -13973.782,E2 -13973.782} C_VEL
LIN {X 0,Y 354.294,Z 235.414,A -85,B 0,C 180,E1 -13975.088,E2 -13975.088} C_VEL
LIN {X 0,Y 355.44,Z 225.083,A -85,B 0,C 180,E1 -13976.101,E2 -13976.101} C_VEL
LIN {X 0,Y 356.665,Z 212.47,A -85,B 0,C 180,E1 -13977.05,E2 -13977.05} C_VEL
LIN {X 0,Y 357.513,Z 199.423,A -85,B 0,C 180,E1 -13977.766,E2 -13977.766} C_VEL
LIN {X 0,Y 357.729,Z 195.765,A -85,B 0,C 180,E1 -13977.919,E2 -13977.919} C_VEL
LIN {X 0,Y 357.491,Z 190.057,A -85,B 0,C 180,E1 -13978.162,E2 -13978.162} C_VEL
LIN {X 0,Y 352.639,Z 171.502,A -85,B 0,C 180,E1 -13978.989,E2 -13978.989} C_VEL
LIN {X 0,Y 352.165,Z 165.695,A -85,B 0,C 180,E1 -13979.149,E2 -13979.149} C_VEL
LIN {X 0,Y 353.424,Z 108.424,A -85,B 0,C 180,E1 -13980.32,E2 -13980.32} C_VEL
LIN {X 0,Y 351.801,Z 103.436,A -85,B 0,C 180,E1 -13980.563,E2 -13980.563} C_VEL
LIN {X 0,Y 344.569,Z 86.556,A -85,B 0,C 180,E1 -13981.555,E2 -13981.555} C_VEL
LIN {X 0,Y 342.013,Z 80.758,A -85,B 0,C 180,E1 -13981.94,E2 -13981.94} C_VEL
LIN {X 0,Y 340.71,Z 75.048,A -85,B 0,C 180,E1 -13983.845,E2 -13983.845} C_VEL
LIN {X 0,Y 340.704,Z 75.044,A -85,B 0,C 180,E1 -13986.742,E2 -13986.742} C_VEL
LIN {X 0,Y 340.654,Z 75.053,A -85,B 0,C 180,E1 -13990.239,E2 -13990.239} C_VEL
LIN {X 0,Y 340.675,Z 75.049,A -85,B 0,C 180,E1 -13992.905,E2 -13992.905} C_VEL
LIN {X 0,Y 340.675,Z 75.049,A -85,B 0,C 180,E1 -13997.095,E2 -13997.095} C_VEL
LIN {X 0,Y 340.658,Z 75.05,A -85,B 0,C 180,E1 -14000.241,E2 -14000.241} C_VEL
LIN {X 0,Y 340.709,Z 75.044,A -85,B 0,C 180,E1 -14003.56,E2 -14003.56} C_VEL
LIN {X 0,Y 340.695,Z 75.046,A -85,B 0,C 180,E1 -14006.153,E2 -14006.153} C_VEL
LIN {X 0,Y 340.72,Z 75.042,A -85,B 0,C 180,E1 -14010.036,E2 -14010.036} C_VEL
LIN {X 0,Y 340.714,Z 75.037,A -85,B 0,C 180,E1 -14013.012,E2 -14013.012} C_VEL
LIN {X 0,Y 340.742,Z 75.038,A -85,B 0,C 180,E1 -14015.637,E2 -14015.637} C_VEL
LIN {X 0,Y 340.737,Z 75.041,A -85,B 0,C 180,E1 -14019.473,E2 -14019.473} C_VEL
LIN {X 0,Y 340.796,Z 75.025,A -85,B 0,C 180,E1 -14021.98,E2 -14021.98} C_VEL
LIN {X 0,Y 340.873,Z 75.022,A -85,B 0,C 180,E1 -14025.705,E2 -14025.705} C_VEL
LIN {X 0,Y 340.851,Z 75.023,A -85,B 0,C 180,E1 -14029.305,E2 -14029.305} C_VEL
LIN {X 0,Y 341.001,Z 74.998,A -85,B 0,C 180,E1 -14032.896,E2 -14032.896} C_VEL
LIN {X 0,Y 340.822,Z 75.026,A -85,B 0,C 180,E1 -14035.268,E2 -14035.268} C_VEL
LIN {X 0,Y 341.133,Z 74.991,A -85,B 0,C 180,E1 -14037.638,E2 -14037.638} C_VEL
LIN {X 0,Y 341.112,Z 74.988,A -85,B 0,C 180,E1 -14041.18,E2 -14041.18} C_VEL
LIN {X 0,Y 341.128,Z 74.994,A -85,B 0,C 180,E1 -14042.361,E2 -14042.361} C_VEL
LIN {X 0,Y 341.018,Z 74.994,A -85,B 0,C 180,E1 -14045.914,E2 -14045.914} C_VEL
LIN {X 0,Y 340.966,Z 75.012,A -85,B 0,C 180,E1 -14048.356,E2 -14048.356} C_VEL
LIN {X 0,Y 340.852,Z 75.015,A -85,B 0,C 180,E1 -14051.899,E2 -14051.899} C_VEL
LIN {X 0,Y 340.82,Z 75.028,A -85,B 0,C 180,E1 -14055.549,E2 -14055.549} C_VEL
LIN {X 0,Y 340.767,Z 75.036,A -85,B 0,C 180,E1 -14059.268,E2 -14059.268} C_VEL
LIN {X 0,Y 340.731,Z 75.034,A -85,B 0,C 180,E1 -14063.073,E2 -14063.073} C_VEL
LIN {X 0,Y 340.775,Z 75.033,A -85,B 0,C 180,E1 -14065.664,E2 -14065.664} C_VEL
LIN {X 0,Y 340.731,Z 75.039,A -85,B 0,C 180,E1 -14068.32,E2 -14068.32} C_VEL
LIN {X 0,Y 340.7,Z 75.04,A -85,B 0,C 180,E1 -14071.044,E2 -14071.044} C_VEL
LIN {X 0,Y 340.72,Z 75.026,A -85,B 0,C 180,E1 -14075.279,E2 -14075.279} C_VEL
LIN {X 0,Y 340.712,Z 75.037,A -85,B 0,C 180,E1 -14078.386,E2 -14078.386} C_VEL
LIN {X 0,Y 340.701,Z 75.044,A -85,B 0,C 180,E1 -14082.045,E2 -14082.045} C_VEL
LIN {X 0,Y 340.654,Z 75.048,A -85,B 0,C 180,E1 -14086.227,E2 -14086.227} C_VEL
LIN {X 0,Y 340.691,Z 75.045,A -85,B 0,C 180,E1 -14089.753,E2 -14089.753} C_VEL
LIN {X 0,Y 340.707,Z 75.045,A -85,B 0,C 180,E1 -14093.258,E2 -14093.258} C_VEL
LIN {X 0,Y 340.73,Z 75.177,A -85,B 0,C 180,E1 -14096.601,E2 -14096.601} C_VEL
LIN {X 0,Y 343.535,Z 86.737,A -85,B 0,C 180,E1 -14099.954,E2 -14099.954} C_VEL
LIN {X 0,Y 345.743,Z 97.056,A -85,B 0,C 180,E1 -14102.783,E2 -14102.783} C_VEL
LIN {X 0,Y 346.166,Z 99.668,A -85,B 0,C 180,E1 -14103.47,E2 -14103.47} C_VEL
LIN {X 0,Y 345.208,Z 107.763,A -85,B 0,C 180,E1 -14105.4,E2 -14105.4} C_VEL
LIN {X 0,Y 350.632,Z 135.905,A -85,B 0,C 180,E1 -14106.492,E2 -14106.492} C_VEL
LIN {X 0,Y 352.577,Z 148.603,A -85,B 0,C 180,E1 -14106.927,E2 -14106.927} C_VEL
LIN {X 0,Y 351.094,Z 216.49,A -85,B 0,C 180,E1 -14108.341,E2 -14108.341} C_VEL
LIN {X 0,Y 350.247,Z 229.745,A -85,B 0,C 180,E1 -14108.827,E2 -14108.827} C_VEL
LIN {X 0,Y 349.034,Z 242.46,A -85,B 0,C 180,E1 -14109.521,E2 -14109.521} C_VEL
LIN {X 0,Y 347.812,Z 253.769,A -85,B 0,C 180,E1 -14110.37,E2 -14110.37} C_VEL
LIN {X 0,Y 346.286,Z 265.437,A -85,B 0,C 180,E1 -14111.511,E2 -14111.511} C_VEL
LIN {X 0,Y 344.736,Z 275.936,A -85,B 0,C 180,E1 -14112.806,E2 -14112.806} C_VEL
LIN {X 0,Y 343.426,Z 284.553,A -85,B 0,C 180,E1 -14114.118,E2 -14114.118} C_VEL
LIN {X 0,Y 342.222,Z 293.208,A -85,B 0,C 180,E1 -14115.733,E2 -14115.733} C_VEL
LIN {X 0,Y 341.01,Z 300.838,A -85,B 0,C 180,E1 -14117.502,E2 -14117.502} C_VEL
LIN {X 0,Y 340.159,Z 306.998,A -85,B 0,C 180,E1 -14119.283,E2 -14119.283} C_VEL
LIN {X 0,Y 339.573,Z 311.906,A -85,B 0,C 180,E1 -14121.07,E2 -14121.07} C_VEL
LIN {X 0,Y 339.247,Z 315.704,A -85,B 0,C 180,E1 -14122.859,E2 -14122.859} C_VEL
LIN {X 0,Y 339.128,Z 317.777,A -85,B 0,C 180,E1 -14124.121,E2 -14124.121} C_VEL
LIN {X 0,Y 339.069,Z 319.229,A -85,B 0,C 180,E1 -14125.244,E2 -14125.244} C_VEL
LIN {X 0,Y 339.085,Z 320.339,A -85,B 0,C 180,E1 -14126.435,E2 -14126.435} C_VEL
LIN {X 0,Y 339.161,Z 321.37,A -85,B 0,C 180,E1 -14128.812,E2 -14128.812} C_VEL
LIN {X 0,Y 339.229,Z 321.306,A -85,B 0,C 180,E1 -14130,E2 -14130} C_VEL
LIN {X 0,Y 339.174,Z 320.807,A -85,B 0,C 180,E1 -14131.187,E2 -14131.187} C_VEL
LIN {X 0,Y 339.122,Z 318.587,A -85,B 0,C 180,E1 -14133.564,E2 -14133.564} C_VEL
LIN {X 0,Y 339.118,Z 316.864,A -85,B 0,C 180,E1 -14134.755,E2 -14134.755} C_VEL
LIN {X 0,Y 339.147,Z 313.39,A -85,B 0,C 180,E1 -14136.544,E2 -14136.544} C_VEL
LIN {X 0,Y 339.407,Z 308.822,A -85,B 0,C 180,E1 -14138.334,E2 -14138.334} C_VEL
LIN {X 0,Y 339.864,Z 301.877,A -85,B 0,C 180,E1 -14140.424,E2 -14140.424} C_VEL
LIN {X 0,Y 340.573,Z 294.347,A -85,B 0,C 180,E1 -14142.211,E2 -14142.211} C_VEL
LIN {X 0,Y 341.313,Z 286.658,A -85,B 0,C 180,E1 -14143.697,E2 -14143.697} C_VEL
LIN {X 0,Y 342.22,Z 277.478,A -85,B 0,C 180,E1 -14145.157,E2 -14145.157} C_VEL
LIN {X 0,Y 343.25,Z 266.92,A -85,B 0,C 180,E1 -14146.504,E2 -14146.504} C_VEL
LIN {X 0,Y 344.432,Z 255.388,A -85,B 0,C 180,E1 -14147.669,E2 -14147.669} C_VEL
LIN {X 0,Y 345.415,Z 243.305,A -85,B 0,C 180,E1 -14148.613,E2 -14148.613} C_VEL
LIN {X 0,Y 346.4,Z 230.635,A -85,B 0,C 180,E1 -14149.327,E2 -14149.327} C_VEL
LIN {X 0,Y 346.951,Z 217.462,A -85,B 0,C 180,E1 -14149.834,E2 -14149.834} C_VEL
LIN {X 0,Y 348.099,Z 145.868,A -85,B 0,C 180,E1 -14151.331,E2 -14151.331} C_VEL
LIN {X 0,Y 343.25,Z 110.214,A -85,B 0,C 180,E1 -14152.373,E2 -14152.373} C_VEL
LIN {X 0,Y 342.96,Z 108.206,A -85,B 0,C 180,E1 -14152.453,E2 -14152.453} C_VEL
LIN {X 0,Y 344.329,Z 94.046,A -85,B 0,C 180,E1 -14155.725,E2 -14155.725} C_VEL
LIN {X 0,Y 343.315,Z 87.223,A -85,B 0,C 180,E1 -14157.425,E2 -14157.425} C_VEL
LIN {X 0,Y 340.75,Z 75.04,A -85,B 0,C 180,E1 -14160.626,E2 -14160.626} C_VEL
LIN {X 0,Y 340.723,Z 75.042,A -85,B 0,C 180,E1 -14164.404,E2 -14164.404} C_VEL
LIN {X 0,Y 340.712,Z 75.042,A -85,B 0,C 180,E1 -14168.386,E2 -14168.386} C_VEL
LIN {X 0,Y 340.698,Z 75.045,A -85,B 0,C 180,E1 -14172.045,E2 -14172.045} C_VEL
LIN {X 0,Y 340.651,Z 75.049,A -85,B 0,C 180,E1 -14176.227,E2 -14176.227} C_VEL
LIN {X 0,Y 340.687,Z 75.046,A -85,B 0,C 180,E1 -14179.753,E2 -14179.753} C_VEL
LIN {X 0,Y 340.704,Z 75.047,A -85,B 0,C 180,E1 -14183.258,E2 -14183.258} C_VEL
LIN {X 0,Y 340.691,Z 75.044,A -85,B 0,C 180,E1 -14186.153,E2 -14186.153} C_VEL
LIN {X 0,Y 340.773,Z 75.034,A -85,B 0,C 180,E1 -14190.332,E2 -14190.332} C_VEL
LIN {X 0,Y 340.803,Z 75.035,A -85,B 0,C 180,E1 -14193.02,E2 -14193.02} C_VEL
LIN {X 0,Y 340.755,Z 75.036,A -85,B 0,C 180,E1 -14195.638,E2 -14195.638} C_VEL
LIN {X 0,Y 340.751,Z 75.036,A -85,B 0,C 180,E1 -14199.475,E2 -14199.475} C_VEL
LIN {X 0,Y 340.857,Z 75.024,A -85,B 0,C 180,E1 -14201.984,E2 -14201.984} C_VEL
LIN {X 0,Y 340.868,Z 75.022,A -85,B 0,C 180,E1 -14205.705,E2 -14205.705} C_VEL
LIN {X 0,Y 340.87,Z 75.021,A -85,B 0,C 180,E1 -14209.306,E2 -14209.306} C_VEL
LIN {X 0,Y 341.058,Z 74.999,A -85,B 0,C 180,E1 -14212.898,E2 -14212.898} C_VEL
LIN {X 0,Y 341.164,Z 74.985,A -85,B 0,C 180,E1 -14217.639,E2 -14217.639} C_VEL
LIN {X 0,Y 341.274,Z 74.976,A -85,B 0,C 180,E1 -14220,E2 -14220} C_VEL
LIN {X 0,Y 341.165,Z 74.987,A -85,B 0,C 180,E1 -14222.362,E2 -14222.362} C_VEL
LIN {X 0,Y 341.018,Z 75.003,A -85,B 0,C 180,E1 -14227.103,E2 -14227.103} C_VEL
LIN {X 0,Y 340.848,Z 75.024,A -85,B 0,C 180,E1 -14230.695,E2 -14230.695} C_VEL
LIN {X 0,Y 340.863,Z 75.022,A -85,B 0,C 180,E1 -14234.325,E2 -14234.325} C_VEL
LIN {X 0,Y 340.837,Z 75.025,A -85,B 0,C 180,E1 -14238.467,E2 -14238.467} C_VEL
LIN {X 0,Y 340.754,Z 75.037,A -85,B 0,C 180,E1 -14241.857,E2 -14241.857} C_VEL
LIN {X 0,Y 340.772,Z 75.036,A -85,B 0,C 180,E1 -14245.665,E2 -14245.665} C_VEL
LIN {X 0,Y 340.729,Z 75.039,A -85,B 0,C 180,E1 -14248.321,E2 -14248.321} C_VEL
LIN {X 0,Y 340.698,Z 75.048,A -85,B 0,C 180,E1 -14251.045,E2 -14251.045} C_VEL
LIN {X 0,Y 340.718,Z 75.044,A -85,B 0,C 180,E1 -14255.279,E2 -14255.279} C_VEL
LIN {X 0,Y 340.694,Z 75.045,A -85,B 0,C 180,E1 -14258.383,E2 -14258.383} C_VEL
LIN {X 0,Y 340.694,Z 75.044,A -85,B 0,C 180,E1 -14262.045,E2 -14262.045} C_VEL
LIN {X 0,Y 340.653,Z 75.051,A -85,B 0,C 180,E1 -14266.228,E2 -14266.228} C_VEL
LIN {X 0,Y 340.675,Z 75.046,A -85,B 0,C 180,E1 -14269.756,E2 -14269.756} C_VEL
LIN {X 0,Y 340.704,Z 75.042,A -85,B 0,C 180,E1 -14273.259,E2 -14273.259} C_VEL
LIN {X 0,Y 340.696,Z 75.048,A -85,B 0,C 180,E1 -14276.154,E2 -14276.154} C_VEL
LIN {X 0,Y 340.726,Z 75.044,A -85,B 0,C 180,E1 -14280.034,E2 -14280.034} C_VEL
LIN {X 0,Y 340.722,Z 75.04,A -85,B 0,C 180,E1 -14283.013,E2 -14283.013} C_VEL
LIN {X 0,Y 340.708,Z 75.042,A -85,B 0,C 180,E1 -14286.926,E2 -14286.926} C_VEL
LIN {X 0,Y 340.794,Z 75.032,A -85,B 0,C 180,E1 -14290.734,E2 -14290.734} C_VEL
LIN {X 0,Y 340.844,Z 75.157,A -85,B 0,C 180,E1 -14293.068,E2 -14293.068} C_VEL
LIN {X 0,Y 341.902,Z 80.516,A -85,B 0,C 180,E1 -14294.593,E2 -14294.593} C_VEL
LIN {X 0,Y 347.325,Z 96.648,A -85,B 0,C 180,E1 -14295.268,E2 -14295.268} C_VEL
LIN {X 0,Y 348.881,Z 105.214,A -85,B 0,C 180,E1 -14295.541,E2 -14295.541} C_VEL
LIN {X 0,Y 347.33,Z 187.703,A -85,B 0,C 180,E1 -14297.251,E2 -14297.251} C_VEL
LIN {X 0,Y 346.871,Z 200.657,A -85,B 0,C 180,E1 -14297.754,E2 -14297.754} C_VEL
LIN {X 0,Y 346.261,Z 212.624,A -85,B 0,C 180,E1 -14298.438,E2 -14298.438} C_VEL
LIN {X 0,Y 345.549,Z 223.933,A -85,B 0,C 180,E1 -14299.305,E2 -14299.305} C_VEL
LIN {X 0,Y 344.558,Z 235.569,A -85,B 0,C 180,E1 -14300.461,E2 -14300.461} C_VEL
LIN {X 0,Y 343.524,Z 246.015,A -85,B 0,C 180,E1 -14301.767,E2 -14301.767} C_VEL
LIN {X 0,Y 342.547,Z 255.436,A -85,B 0,C 180,E1 -14303.225,E2 -14303.225} C_VEL
LIN {X 0,Y 341.484,Z 264.511,A -85,B 0,C 180,E1 -14304.982,E2 -14304.982} C_VEL
LIN {X 0,Y 340.709,Z 271.814,A -85,B 0,C 180,E1 -14306.748,E2 -14306.748} C_VEL
LIN {X 0,Y 340.015,Z 278.537,A -85,B 0,C 180,E1 -14308.816,E2 -14308.816} C_VEL
LIN {X 0,Y 339.629,Z 282.976,A -85,B 0,C 180,E1 -14310.593,E2 -14310.593} C_VEL
LIN {X 0,Y 339.381,Z 286.354,A -85,B 0,C 180,E1 -14312.374,E2 -14312.374} C_VEL
LIN {X 0,Y 339.238,Z 289.318,A -85,B 0,C 180,E1 -14314.754,E2 -14314.754} C_VEL
LIN {X 0,Y 339.294,Z 290.315,A -85,B 0,C 180,E1 -14316.14,E2 -14316.14} C_VEL
LIN {X 0,Y 339.173,Z 290.764,A -85,B 0,C 180,E1 -14318.34,E2 -14318.34} C_VEL
LIN {X 0,Y 339.278,Z 289.759,A -85,B 0,C 180,E1 -14320.745,E2 -14320.745} C_VEL
LIN {X 0,Y 339.535,Z 288.625,A -85,B 0,C 180,E1 -14321.946,E2 -14321.946} C_VEL
LIN {X 0,Y 339.978,Z 286.254,A -85,B 0,C 180,E1 -14323.69,E2 -14323.69} C_VEL
LIN {X 0,Y 340.517,Z 282.65,A -85,B 0,C 180,E1 -14325.564,E2 -14325.564} C_VEL
LIN {X 0,Y 341.312,Z 278.017,A -85,B 0,C 180,E1 -14327.372,E2 -14327.372} C_VEL
LIN {X 0,Y 342.439,Z 270.983,A -85,B 0,C 180,E1 -14329.482,E2 -14329.482} C_VEL
LIN {X 0,Y 343.722,Z 263.322,A -85,B 0,C 180,E1 -14331.281,E2 -14331.281} C_VEL
LIN {X 0,Y 345.215,Z 253.799,A -85,B 0,C 180,E1 -14333.043,E2 -14333.043} C_VEL
LIN {X 0,Y 346.629,Z 243.57,A -85,B 0,C 180,E1 -14334.56,E2 -14334.56} C_VEL
LIN {X 0,Y 347.919,Z 233.567,A -85,B 0,C 180,E1 -14335.741,E2 -14335.741} C_VEL
LIN {X 0,Y 349.196,Z 222.638,A -85,B 0,C 180,E1 -14336.765,E2 -14336.765} C_VEL
LIN {X 0,Y 350.337,Z 210.355,A -85,B 0,C 180,E1 -14337.652,E2 -14337.652} C_VEL
LIN {X 0,Y 351.137,Z 198.164,A -85,B 0,C 180,E1 -14338.298,E2 -14338.298} C_VEL
LIN {X 0,Y 351.741,Z 184.633,A -85,B 0,C 180,E1 -14338.751,E2 -14338.751} C_VEL
LIN {X 0,Y 352.165,Z 165.695,A -85,B 0,C 180,E1 -14339.149,E2 -14339.149} C_VEL
LIN {X 0,Y 351.637,Z 161.817,A -85,B 0,C 180,E1 -14339.276,E2 -14339.276} C_VEL
LIN {X 0,Y 346.662,Z 149.895,A -85,B 0,C 180,E1 -14339.933,E2 -14339.933} C_VEL
LIN {X 0,Y 346.188,Z 146.018,A -85,B 0,C 180,E1 -14340.059,E2 -14340.059} C_VEL
LIN {X 0,Y 346.997,Z 109.533,A -85,B 0,C 180,E1 -14340.821,E2 -14340.821} C_VEL
LIN {X 0,Y 340.78,Z 94.06,A -85,B 0,C 180,E1 -14341.712,E2 -14341.712} C_VEL
LIN {X 0,Y 334.858,Z 81.068,A -85,B 0,C 180,E1 -14342.597,E2 -14342.597} C_VEL
LIN {X 0,Y 333.681,Z 75.919,A -85,B 0,C 180,E1 -14344.384,E2 -14344.384} C_VEL
LIN {X 0,Y 333.646,Z 75.919,A -85,B 0,C 180,E1 -14347.652,E2 -14347.652} C_VEL
LIN {X 0,Y 333.606,Z 75.93,A -85,B 0,C 180,E1 -14350.774,E2 -14350.774} C_VEL
LIN {X 0,Y 333.592,Z 75.917,A -85,B 0,C 180,E1 -14354.249,E2 -14354.249} C_VEL
LIN {X 0,Y 333.638,Z 75.926,A -85,B 0,C 180,E1 -14357.617,E2 -14357.617} C_VEL
LIN {X 0,Y 333.618,Z 75.925,A -85,B 0,C 180,E1 -14361.21,E2 -14361.21} C_VEL
LIN {X 0,Y 333.676,Z 75.918,A -85,B 0,C 180,E1 -14363.86,E2 -14363.86} C_VEL
LIN {X 0,Y 333.643,Z 75.922,A -85,B 0,C 180,E1 -14367.414,E2 -14367.414} C_VEL
LIN {X 0,Y 333.651,Z 75.925,A -85,B 0,C 180,E1 -14371.022,E2 -14371.022} C_VEL
LIN {X 0,Y 333.697,Z 75.92,A -85,B 0,C 180,E1 -14375.088,E2 -14375.088} C_VEL
LIN {X 0,Y 333.67,Z 75.921,A -85,B 0,C 180,E1 -14379.018,E2 -14379.018} C_VEL
LIN {X 0,Y 333.745,Z 75.904,A -85,B 0,C 180,E1 -14381.586,E2 -14381.586} C_VEL
LIN {X 0,Y 333.812,Z 75.902,A -85,B 0,C 180,E1 -14385.577,E2 -14385.577} C_VEL
LIN {X 0,Y 333.82,Z 75.897,A -85,B 0,C 180,E1 -14389.077,E2 -14389.077} C_VEL
LIN {X 0,Y 333.957,Z 75.876,A -85,B 0,C 180,E1 -14392.746,E2 -14392.746} C_VEL
LIN {X 0,Y 333.787,Z 75.902,A -85,B 0,C 180,E1 -14395.168,E2 -14395.168} C_VEL
LIN {X 0,Y 334.074,Z 75.87,A -85,B 0,C 180,E1 -14397.588,E2 -14397.588} C_VEL
LIN {X 0,Y 334.081,Z 75.864,A -85,B 0,C 180,E1 -14401.205,E2 -14401.205} C_VEL
LIN {X 0,Y 333.807,Z 75.905,A -85,B 0,C 180,E1 -14403.621,E2 -14403.621} C_VEL
LIN {X 0,Y 333.991,Z 75.869,A -85,B 0,C 180,E1 -14406.039,E2 -14406.039} C_VEL
LIN {X 0,Y 333.823,Z 75.901,A -85,B 0,C 180,E1 -14409.696,E2 -14409.696} C_VEL
LIN {X 0,Y 333.8,Z 75.899,A -85,B 0,C 180,E1 -14413.391,E2 -14413.391} C_VEL
LIN {X 0,Y 333.721,Z 75.904,A -85,B 0,C 180,E1 -14417.147,E2 -14417.147} C_VEL
LIN {X 0,Y 333.724,Z 75.916,A -85,B 0,C 180,E1 -14419.691,E2 -14419.691} C_VEL
LIN {X 0,Y 333.695,Z 75.907,A -85,B 0,C 180,E1 -14422.278,E2 -14422.278} C_VEL
LIN {X 0,Y 333.737,Z 75.907,A -85,B 0,C 180,E1 -14426.246,E2 -14426.246} C_VEL
LIN {X 0,Y 333.693,Z 75.92,A -85,B 0,C 180,E1 -14428.974,E2 -14428.974} C_VEL
LIN {X 0,Y 333.646,Z 75.923,A -85,B 0,C 180,E1 -14432.587,E2 -14432.587} C_VEL
LIN {X 0,Y 333.678,Z 75.896,A -85,B 0,C 180,E1 -14436.139,E2 -14436.139} C_VEL
LIN {X 0,Y 333.649,Z 75.926,A -85,B 0,C 180,E1 -14439.192,E2 -14439.192} C_VEL
LIN {X 0,Y 333.635,Z 75.928,A -85,B 0,C 180,E1 -14442.5,E2 -14442.5} C_VEL
LIN {X 0,Y 333.598,Z 75.927,A -85,B 0,C 180,E1 -14445.955,E2 -14445.955} C_VEL
LIN {X 0,Y 333.649,Z 75.921,A -85,B 0,C 180,E1 -14449.315,E2 -14449.315} C_VEL
LIN {X 0,Y 333.667,Z 75.922,A -85,B 0,C 180,E1 -14453.167,E2 -14453.167} C_VEL
LIN {X 0,Y 333.695,Z 76.115,A -85,B 0,C 180,E1 -14456.074,E2 -14456.074} C_VEL
LIN {X 0,Y 336.281,Z 86.816,A -85,B 0,C 180,E1 -14459.273,E2 -14459.273} C_VEL
LIN {X 0,Y 338.557,Z 96.993,A -85,B 0,C 180,E1 -14462.155,E2 -14462.155} C_VEL
LIN {X 0,Y 339.266,Z 100.983,A -85,B 0,C 180,E1 -14463.239,E2 -14463.239} C_VEL
LIN {X 0,Y 338.532,Z 107.414,A -85,B 0,C 180,E1 -14464.811,E2 -14464.811} C_VEL
LIN {X 0,Y 344.171,Z 136.599,A -85,B 0,C 180,E1 -14465.984,E2 -14465.984} C_VEL
LIN {X 0,Y 346.186,Z 149.502,A -85,B 0,C 180,E1 -14466.442,E2 -14466.442} C_VEL
LIN {X 0,Y 344.608,Z 216.767,A -85,B 0,C 180,E1 -14467.873,E2 -14467.873} C_VEL
LIN {X 0,Y 343.68,Z 230.58,A -85,B 0,C 180,E1 -14468.402,E2 -14468.402} C_VEL
LIN {X 0,Y 342.427,Z 242.981,A -85,B 0,C 180,E1 -14469.108,E2 -14469.108} C_VEL
LIN {X 0,Y 340.952,Z 255.632,A -85,B 0,C 180,E1 -14470.116,E2 -14470.116} C_VEL
LIN {X 0,Y 339.36,Z 266.894,A -85,B 0,C 180,E1 -14471.276,E2 -14471.276} C_VEL
LIN {X 0,Y 337.784,Z 277.066,A -85,B 0,C 180,E1 -14472.597,E2 -14472.597} C_VEL
LIN {X 0,Y 336.513,Z 285.138,A -85,B 0,C 180,E1 -14473.884,E2 -14473.884} C_VEL
LIN {X 0,Y 335.135,Z 294.502,A -85,B 0,C 180,E1 -14475.735,E2 -14475.735} C_VEL
LIN {X 0,Y 333.86,Z 301.845,A -85,B 0,C 180,E1 -14477.539,E2 -14477.539} C_VEL
LIN {X 0,Y 332.905,Z 308.612,A -85,B 0,C 180,E1 -14479.662,E2 -14479.662} C_VEL
LIN {X 0,Y 332.373,Z 313.101,A -85,B 0,C 180,E1 -14481.488,E2 -14481.488} C_VEL
LIN {X 0,Y 332.174,Z 315.48,A -85,B 0,C 180,E1 -14482.706,E2 -14482.706} C_VEL
LIN {X 0,Y 332.027,Z 317.805,A -85,B 0,C 180,E1 -14484.181,E2 -14484.181} C_VEL
LIN {X 0,Y 332.008,Z 320.055,A -85,B 0,C 180,E1 -14486.359,E2 -14486.359} C_VEL
LIN {X 0,Y 332.063,Z 321.057,A -85,B 0,C 180,E1 -14488.787,E2 -14488.787} C_VEL
LIN {X 0,Y 332.136,Z 320.974,A -85,B 0,C 180,E1 -14490,E2 -14490} C_VEL
LIN {X 0,Y 332.078,Z 320.45,A -85,B 0,C 180,E1 -14491.212,E2 -14491.212} C_VEL
LIN {X 0,Y 332.044,Z 318.2,A -85,B 0,C 180,E1 -14493.64,E2 -14493.64} C_VEL
LIN {X 0,Y 332.007,Z 314.805,A -85,B 0,C 180,E1 -14495.785,E2 -14495.785} C_VEL
LIN {X 0,Y 332.241,Z 309.985,A -85,B 0,C 180,E1 -14497.903,E2 -14497.903} C_VEL
LIN {X 0,Y 332.642,Z 303.537,A -85,B 0,C 180,E1 -14500.038,E2 -14500.038} C_VEL
LIN {X 0,Y 333.276,Z 296.502,A -85,B 0,C 180,E1 -14501.865,E2 -14501.865} C_VEL
LIN {X 0,Y 334.178,Z 287.674,A -85,B 0,C 180,E1 -14503.685,E2 -14503.685} C_VEL
LIN {X 0,Y 335.155,Z 279.198,A -85,B 0,C 180,E1 -14505.107,E2 -14505.107} C_VEL
LIN {X 0,Y 336.073,Z 268.663,A -85,B 0,C 180,E1 -14506.554,E2 -14506.554} C_VEL
LIN {X 0,Y 337.308,Z 257.657,A -85,B 0,C 180,E1 -14507.741,E2 -14507.741} C_VEL
LIN {X 0,Y 338.423,Z 245.287,A -85,B 0,C 180,E1 -14508.777,E2 -14508.777} C_VEL
LIN {X 0,Y 339.316,Z 233.587,A -85,B 0,C 180,E1 -14509.511,E2 -14509.511} C_VEL
LIN {X 0,Y 340.081,Z 221.167,A -85,B 0,C 180,E1 -14510.055,E2 -14510.055} C_VEL
LIN {X 0,Y 340.46,Z 207.05,A -85,B 0,C 180,E1 -14510.425,E2 -14510.425} C_VEL
LIN {X 0,Y 341.334,Z 146.079,A -85,B 0,C 180,E1 -14511.703,E2 -14511.703} C_VEL
LIN {X 0,Y 336.09,Z 107.922,A -85,B 0,C 180,E1 -14512.864,E2 -14512.864} C_VEL
LIN {X 0,Y 337.385,Z 94.892,A -85,B 0,C 180,E1 -14515.941,E2 -14515.941} C_VEL
LIN {X 0,Y 335.72,Z 85.154,A -85,B 0,C 180,E1 -14518.45,E2 -14518.45} C_VEL
LIN {X 0,Y 333.681,Z 75.92,A -85,B 0,C 180,E1 -14520.977,E2 -14520.977} C_VEL
LIN {X 0,Y 333.685,Z 75.918,A -85,B 0,C 180,E1 -14524.774,E2 -14524.774} C_VEL
LIN {X 0,Y 333.654,Z 75.927,A -85,B 0,C 180,E1 -14527.65,E2 -14527.65} C_VEL
LIN {X 0,Y 333.646,Z 75.922,A -85,B 0,C 180,E1 -14530.767,E2 -14530.767} C_VEL
LIN {X 0,Y 333.592,Z 75.929,A -85,B 0,C 180,E1 -14534.25,E2 -14534.25} C_VEL
LIN {X 0,Y 333.64,Z 75.926,A -85,B 0,C 180,E1 -14537.618,E2 -14537.618} C_VEL
LIN {X 0,Y 333.651,Z 75.923,A -85,B 0,C 180,E1 -14541.202,E2 -14541.202} C_VEL
LIN {X 0,Y 333.675,Z 75.918,A -85,B 0,C 180,E1 -14543.861,E2 -14543.861} C_VEL
LIN {X 0,Y 333.642,Z 75.925,A -85,B 0,C 180,E1 -14547.413,E2 -14547.413} C_VEL
LIN {X 0,Y 333.71,Z 75.919,A -85,B 0,C 180,E1 -14551.028,E2 -14551.028} C_VEL
LIN {X 0,Y 333.734,Z 75.91,A -85,B 0,C 180,E1 -14553.754,E2 -14553.754} C_VEL
LIN {X 0,Y 333.718,Z 75.912,A -85,B 0,C 180,E1 -14557.914,E2 -14557.914} C_VEL
LIN {X 0,Y 333.792,Z 75.903,A -85,B 0,C 180,E1 -14561.59,E2 -14561.59} C_VEL
LIN {X 0,Y 333.807,Z 75.901,A -85,B 0,C 180,E1 -14565.577,E2 -14565.577} C_VEL
LIN {X 0,Y 333.833,Z 75.898,A -85,B 0,C 180,E1 -14569.078,E2 -14569.078} C_VEL
LIN {X 0,Y 334.005,Z 75.879,A -85,B 0,C 180,E1 -14572.747,E2 -14572.747} C_VEL
LIN {X 0,Y 333.802,Z 75.901,A -85,B 0,C 180,E1 -14575.169,E2 -14575.169} C_VEL
LIN {X 0,Y 334.101,Z 75.865,A -85,B 0,C 180,E1 -14577.589,E2 -14577.589} C_VEL
LIN {X 0,Y 334.225,Z 75.854,A -85,B 0,C 180,E1 -14580,E2 -14580} C_VEL
LIN {X 0,Y 334.102,Z 75.866,A -85,B 0,C 180,E1 -14582.411,E2 -14582.411} C_VEL
LIN {X 0,Y 333.971,Z 75.881,A -85,B 0,C 180,E1 -14586.493,E2 -14586.493} C_VEL
LIN {X 0,Y 333.82,Z 75.905,A -85,B 0,C 180,E1 -14589.697,E2 -14589.697} C_VEL
LIN {X 0,Y 333.796,Z 75.904,A -85,B 0,C 180,E1 -14593.392,E2 -14593.392} C_VEL
LIN {X 0,Y 333.746,Z 75.911,A -85,B 0,C 180,E1 -14597.147,E2 -14597.147} C_VEL
LIN {X 0,Y 333.736,Z 75.912,A -85,B 0,C 180,E1 -14599.691,E2 -14599.691} C_VEL
LIN {X 0,Y 333.693,Z 75.914,A -85,B 0,C 180,E1 -14602.279,E2 -14602.279} C_VEL
LIN {X 0,Y 333.735,Z 75.91,A -85,B 0,C 180,E1 -14606.247,E2 -14606.247} C_VEL
LIN {X 0,Y 333.69,Z 75.92,A -85,B 0,C 180,E1 -14608.975,E2 -14608.975} C_VEL
LIN {X 0,Y 333.644,Z 75.923,A -85,B 0,C 180,E1 -14612.588,E2 -14612.588} C_VEL
LIN {X 0,Y 333.676,Z 75.918,A -85,B 0,C 180,E1 -14616.14,E2 -14616.14} C_VEL
LIN {X 0,Y 333.62,Z 75.928,A -85,B 0,C 180,E1 -14619.197,E2 -14619.197} C_VEL
LIN {X 0,Y 333.629,Z 75.927,A -85,B 0,C 180,E1 -14622.5,E2 -14622.5} C_VEL
LIN {X 0,Y 333.597,Z 75.928,A -85,B 0,C 180,E1 -14625.955,E2 -14625.955} C_VEL
LIN {X 0,Y 333.644,Z 75.922,A -85,B 0,C 180,E1 -14629.317,E2 -14629.317} C_VEL
LIN {X 0,Y 333.664,Z 75.92,A -85,B 0,C 180,E1 -14633.169,E2 -14633.169} C_VEL
LIN {X 0,Y 333.641,Z 75.923,A -85,B 0,C 180,E1 -14636.792,E2 -14636.792} C_VEL
LIN {X 0,Y 333.664,Z 75.921,A -85,B 0,C 180,E1 -14639.723,E2 -14639.723} C_VEL
LIN {X 0,Y 333.671,Z 75.922,A -85,B 0,C 180,E1 -14642.395,E2 -14642.395} C_VEL
LIN {X 0,Y 333.648,Z 75.924,A -85,B 0,C 180,E1 -14646.409,E2 -14646.409} C_VEL
LIN {X 0,Y 333.736,Z 75.914,A -85,B 0,C 180,E1 -14650.31,E2 -14650.31} C_VEL
LIN {X 0,Y 333.813,Z 76.079,A -85,B 0,C 180,E1 -14652.779,E2 -14652.779} C_VEL
LIN {X 0,Y 334.757,Z 80.764,A -85,B 0,C 180,E1 -14654.152,E2 -14654.152} C_VEL
LIN {X 0,Y 340.82,Z 98.614,A -85,B 0,C 180,E1 -14654.925,E2 -14654.925} C_VEL
LIN {X 0,Y 342.185,Z 106.712,A -85,B 0,C 180,E1 -14655.184,E2 -14655.184} C_VEL
LIN {X 0,Y 340.58,Z 187.413,A -85,B 0,C 180,E1 -14656.88,E2 -14656.88} C_VEL
LIN {X 0,Y 340.118,Z 200.564,A -85,B 0,C 180,E1 -14657.394,E2 -14657.394} C_VEL
LIN {X 0,Y 339.438,Z 213.201,A -85,B 0,C 180,E1 -14658.127,E2 -14658.127} C_VEL
LIN {X 0,Y 338.653,Z 225.232,A -85,B 0,C 180,E1 -14659.084,E2 -14659.084} C_VEL
LIN {X 0,Y 337.63,Z 236.674,A -85,B 0,C 180,E1 -14660.263,E2 -14660.263} C_VEL
LIN {X 0,Y 336.549,Z 246.988,A -85,B 0,C 180,E1 -14661.595,E2 -14661.595} C_VEL
LIN {X 0,Y 335.546,Z 256.271,A -85,B 0,C 180,E1 -14663.083,E2 -14663.083} C_VEL
LIN {X 0,Y 334.435,Z 265.246,A -85,B 0,C 180,E1 -14664.876,E2 -14664.876} C_VEL
LIN {X 0,Y 333.638,Z 272.477,A -85,B 0,C 180,E1 -14666.679,E2 -14666.679} C_VEL
LIN {X 0,Y 332.955,Z 279.103,A -85,B 0,C 180,E1 -14668.791,E2 -14668.791} C_VEL
LIN {X 0,Y 332.544,Z 283.486,A -85,B 0,C 180,E1 -14670.606,E2 -14670.606} C_VEL
LIN {X 0,Y 332.277,Z 286.813,A -85,B 0,C 180,E1 -14672.425,E2 -14672.425} C_VEL
LIN {X 0,Y 332.155,Z 289.725,A -85,B 0,C 180,E1 -14674.855,E2 -14674.855} C_VEL
LIN {X 0,Y 332.221,Z 290.616,A -85,B 0,C 180,E1 -14676.134,E2 -14676.134} C_VEL
LIN {X 0,Y 332.076,Z 291.075,A -85,B 0,C 180,E1 -14678.52,E2 -14678.52} C_VEL
LIN {X 0,Y 332.13,Z 290.74,A -85,B 0,C 180,E1 -14679.747,E2 -14679.747} C_VEL
LIN {X 0,Y 332.232,Z 290.013,A -85,B 0,C 180,E1 -14680.976,E2 -14680.976} C_VEL
LIN {X 0,Y 332.511,Z 288.835,A -85,B 0,C 180,E1 -14682.203,E2 -14682.203} C_VEL
LIN {X 0,Y 332.945,Z 286.668,A -85,B 0,C 180,E1 -14683.831,E2 -14683.831} C_VEL
LIN {X 0,Y 333.56,Z 282.752,A -85,B 0,C 180,E1 -14685.897,E2 -14685.897} C_VEL
LIN {X 0,Y 334.409,Z 278.059,A -85,B 0,C 180,E1 -14687.743,E2 -14687.743} C_VEL
LIN {X 0,Y 335.61,Z 270.959,A -85,B 0,C 180,E1 -14689.895,E2 -14689.895} C_VEL
LIN {X 0,Y 337.001,Z 263.191,A -85,B 0,C 180,E1 -14691.726,E2 -14691.726} C_VEL
LIN {X 0,Y 338.547,Z 253.778,A -85,B 0,C 180,E1 -14693.486,E2 -14693.486} C_VEL
LIN {X 0,Y 339.912,Z 244.312,A -85,B 0,C 180,E1 -14694.915,E2 -14694.915} C_VEL
LIN {X 0,Y 341.244,Z 234.436,A -85,B 0,C 180,E1 -14696.119,E2 -14696.119} C_VEL
LIN {X 0,Y 342.573,Z 223.653,A -85,B 0,C 180,E1 -14697.16,E2 -14697.16} C_VEL
LIN {X 0,Y 343.837,Z 210.722,A -85,B 0,C 180,E1 -14698.116,E2 -14698.116} C_VEL
LIN {X 0,Y 344.684,Z 198.406,A -85,B 0,C 180,E1 -14698.779,E2 -14698.779} C_VEL
LIN {X 0,Y 345.31,Z 184.787,A -85,B 0,C 180,E1 -14699.24,E2 -14699.24} C_VEL
LIN {X 0,Y 346.188,Z 146.018,A -85,B 0,C 180,E1 -14700.059,E2 -14700.059} C_VEL
LIN {X 0,Y 345.809,Z 140.21,A -85,B 0,C 180,E1 -14700.222,E2 -14700.222} C_VEL
LIN {X 0,Y 341.072,Z 121.568,A -85,B 0,C 180,E1 -14701.046,E2 -14701.046} C_VEL
LIN {X 0,Y 340.605,Z 115.76,A -85,B 0,C 180,E1 -14701.221,E2 -14701.221} C_VEL
LIN {X 0,Y 340.56,Z 110.853,A -85,B 0,C 180,E1 -14701.34,E2 -14701.34} C_VEL
LIN {X 0,Y 334.225,Z 95.608,A -85,B 0,C 180,E1 -14702.269,E2 -14702.269} C_VEL
LIN {X 0,Y 327.73,Z 81.511,A -85,B 0,C 180,E1 -14703.244,E2 -14703.244} C_VEL
LIN {X 0,Y 326.644,Z 76.794,A -85,B 0,C 180,E1 -14704.902,E2 -14704.902} C_VEL
LIN {X 0,Y 326.585,Z 76.806,A -85,B 0,C 180,E1 -14708.615,E2 -14708.615} C_VEL
LIN {X 0,Y 326.575,Z 76.806,A -85,B 0,C 180,E1 -14712.971,E2 -14712.971} C_VEL
LIN {X 0,Y 326.575,Z 76.805,A -85,B 0,C 180,E1 -14717.029,E2 -14717.029} C_VEL
LIN {X 0,Y 326.574,Z 76.804,A -85,B 0,C 180,E1 -14720.782,E2 -14720.782} C_VEL
LIN {X 0,Y 326.613,Z 76.795,A -85,B 0,C 180,E1 -14724.48,E2 -14724.48} C_VEL
LIN {X 0,Y 326.607,Z 76.798,A -85,B 0,C 180,E1 -14727.455,E2 -14727.455} C_VEL
LIN {X 0,Y 326.59,Z 76.802,A -85,B 0,C 180,E1 -14730.333,E2 -14730.333} C_VEL
LIN {X 0,Y 326.636,Z 76.796,A -85,B 0,C 180,E1 -14734.511,E2 -14734.511} C_VEL
LIN {X 0,Y 326.619,Z 76.794,A -85,B 0,C 180,E1 -14738.543,E2 -14738.543} C_VEL
LIN {X 0,Y 326.711,Z 76.782,A -85,B 0,C 180,E1 -14741.175,E2 -14741.175} C_VEL
LIN {X 0,Y 326.767,Z 76.78,A -85,B 0,C 180,E1 -14745.433,E2 -14745.433} C_VEL
LIN {X 0,Y 326.761,Z 76.773,A -85,B 0,C 180,E1 -14748.838,E2 -14748.838} C_VEL
LIN {X 0,Y 326.914,Z 76.755,A -85,B 0,C 180,E1 -14752.589,E2 -14752.589} C_VEL
LIN {X 0,Y 326.755,Z 76.778,A -85,B 0,C 180,E1 -14755.064,E2 -14755.064} C_VEL
LIN {X 0,Y 327.017,Z 76.749,A -85,B 0,C 180,E1 -14757.536,E2 -14757.536} C_VEL
LIN {X 0,Y 327.048,Z 76.74,A -85,B 0,C 180,E1 -14761.231,E2 -14761.231} C_VEL
LIN {X 0,Y 326.756,Z 76.784,A -85,B 0,C 180,E1 -14763.699,E2 -14763.699} C_VEL
LIN {X 0,Y 326.945,Z 76.746,A -85,B 0,C 180,E1 -14766.17,E2 -14766.17} C_VEL
LIN {X 0,Y 326.786,Z 76.775,A -85,B 0,C 180,E1 -14769.907,E2 -14769.907} C_VEL
LIN {X 0,Y 326.762,Z 76.779,A -85,B 0,C 180,E1 -14773.685,E2 -14773.685} C_VEL
LIN {X 0,Y 326.666,Z 76.783,A -85,B 0,C 180,E1 -14777.53,E2 -14777.53} C_VEL
LIN {X 0,Y 326.657,Z 76.793,A -85,B 0,C 180,E1 -14780.135,E2 -14780.135} C_VEL
LIN {X 0,Y 326.655,Z 76.794,A -85,B 0,C 180,E1 -14784.128,E2 -14784.128} C_VEL
LIN {X 0,Y 326.685,Z 76.784,A -85,B 0,C 180,E1 -14786.857,E2 -14786.857} C_VEL
LIN {X 0,Y 326.636,Z 76.793,A -85,B 0,C 180,E1 -14790.609,E2 -14790.609} C_VEL
LIN {X 0,Y 326.609,Z 76.798,A -85,B 0,C 180,E1 -14794.019,E2 -14794.019} C_VEL
LIN {X 0,Y 326.63,Z 76.777,A -85,B 0,C 180,E1 -14797.238,E2 -14797.238} C_VEL
LIN {X 0,Y 326.58,Z 76.802,A -85,B 0,C 180,E1 -14801.131,E2 -14801.131} C_VEL
LIN {X 0,Y 326.529,Z 76.812,A -85,B 0,C 180,E1 -14804.743,E2 -14804.743} C_VEL
LIN {X 0,Y 326.578,Z 76.801,A -85,B 0,C 180,E1 -14808.154,E2 -14808.154} C_VEL
LIN {X 0,Y 326.626,Z 76.797,A -85,B 0,C 180,E1 -14811.391,E2 -14811.391} C_VEL
LIN {X 0,Y 326.651,Z 76.89,A -85,B 0,C 180,E1 -14815.473,E2 -14815.473} C_VEL
LIN {X 0,Y 329.155,Z 87.216,A -85,B 0,C 180,E1 -14818.657,E2 -14818.657} C_VEL
LIN {X 0,Y 331.369,Z 96.93,A -85,B 0,C 180,E1 -14821.497,E2 -14821.497} C_VEL
LIN {X 0,Y 332.411,Z 102.989,A -85,B 0,C 180,E1 -14823.183,E2 -14823.183} C_VEL
LIN {X 0,Y 331.875,Z 107.095,A -85,B 0,C 180,E1 -14824.205,E2 -14824.205} C_VEL
LIN {X 0,Y 337.382,Z 134.932,A -85,B 0,C 180,E1 -14825.37,E2 -14825.37} C_VEL
LIN {X 0,Y 339.784,Z 150.96,A -85,B 0,C 180,E1 -14825.949,E2 -14825.949} C_VEL
LIN {X 0,Y 338.207,Z 215.927,A -85,B 0,C 180,E1 -14827.351,E2 -14827.351} C_VEL
LIN {X 0,Y 337.279,Z 229.155,A -85,B 0,C 180,E1 -14827.85,E2 -14827.85} C_VEL
LIN {X 0,Y 335.955,Z 242.411,A -85,B 0,C 180,E1 -14828.605,E2 -14828.605} C_VEL
LIN {X 0,Y 334.502,Z 254.339,A -85,B 0,C 180,E1 -14829.555,E2 -14829.555} C_VEL
LIN {X 0,Y 332.869,Z 265.776,A -85,B 0,C 180,E1 -14830.737,E2 -14830.737} C_VEL
LIN {X 0,Y 331.195,Z 276.104,A -85,B 0,C 180,E1 -14832.079,E2 -14832.079} C_VEL
LIN {X 0,Y 329.58,Z 285.751,A -85,B 0,C 180,E1 -14833.655,E2 -14833.655} C_VEL
LIN {X 0,Y 328.215,Z 294.437,A -85,B 0,C 180,E1 -14835.427,E2 -14835.427} C_VEL
LIN {X 0,Y 326.926,Z 301.735,A -85,B 0,C 180,E1 -14837.27,E2 -14837.27} C_VEL
LIN {X 0,Y 326.11,Z 306.692,A -85,B 0,C 180,E1 -14838.816,E2 -14838.816} C_VEL
LIN {X 0,Y 325.494,Z 311.528,A -85,B 0,C 180,E1 -14840.68,E2 -14840.68} C_VEL
LIN {X 0,Y 325.091,Z 315.257,A -85,B 0,C 180,E1 -14842.547,E2 -14842.547} C_VEL
LIN {X 0,Y 324.921,Z 317.79,A -85,B 0,C 180,E1 -14844.253,E2 -14844.253} C_VEL
LIN {X 0,Y 324.932,Z 319.771,A -85,B 0,C 180,E1 -14846.279,E2 -14846.279} C_VEL
LIN {X 0,Y 324.965,Z 320.743,A -85,B 0,C 180,E1 -14848.76,E2 -14848.76} C_VEL
LIN {X 0,Y 325.043,Z 320.638,A -85,B 0,C 180,E1 -14850,E2 -14850} C_VEL
LIN {X 0,Y 324.982,Z 320.091,A -85,B 0,C 180,E1 -14851.239,E2 -14851.239} C_VEL
LIN {X 0,Y 324.967,Z 317.812,A -85,B 0,C 180,E1 -14853.72,E2 -14853.72} C_VEL
LIN {X 0,Y 324.91,Z 314.71,A -85,B 0,C 180,E1 -14855.727,E2 -14855.727} C_VEL
LIN {X 0,Y 325.079,Z 311.062,A -85,B 0,C 180,E1 -14857.453,E2 -14857.453} C_VEL
LIN {X 0,Y 325.377,Z 306.02,A -85,B 0,C 180,E1 -14859.322,E2 -14859.322} C_VEL
LIN {X 0,Y 325.864,Z 299.675,A -85,B 0,C 180,E1 -14861.192,E2 -14861.192} C_VEL
LIN {X 0,Y 326.786,Z 291.732,A -85,B 0,C 180,E1 -14863.051,E2 -14863.051} C_VEL
LIN {X 0,Y 327.706,Z 283.623,A -85,B 0,C 180,E1 -14864.595,E2 -14864.595} C_VEL
LIN {X 0,Y 328.647,Z 273.705,A -85,B 0,C 180,E1 -14866.141,E2 -14866.141} C_VEL
LIN {X 0,Y 329.707,Z 263.989,A -85,B 0,C 180,E1 -14867.363,E2 -14867.363} C_VEL
LIN {X 0,Y 330.873,Z 253.538,A -85,B 0,C 180,E1 -14868.418,E2 -14868.418} C_VEL
LIN {X 0,Y 331.934,Z 240.945,A -85,B 0,C 180,E1 -14869.399,E2 -14869.399} C_VEL
LIN {X 0,Y 332.955,Z 227.668,A -85,B 0,C 180,E1 -14870.14,E2 -14870.14} C_VEL
LIN {X 0,Y 333.461,Z 215.572,A -85,B 0,C 180,E1 -14870.591,E2 -14870.591} C_VEL
LIN {X 0,Y 334.633,Z 146.961,A -85,B 0,C 180,E1 -14872.071,E2 -14872.071} C_VEL
LIN {X 0,Y 329.949,Z 112.678,A -85,B 0,C 180,E1 -14873.129,E2 -14873.129} C_VEL
LIN {X 0,Y 329.265,Z 107.542,A -85,B 0,C 180,E1 -14873.315,E2 -14873.315} C_VEL
LIN {X 0,Y 330.404,Z 97.012,A -85,B 0,C 180,E1 -14875.852,E2 -14875.852} C_VEL
LIN {X 0,Y 329.723,Z 91.497,A -85,B 0,C 180,E1 -14877.274,E2 -14877.274} C_VEL
LIN {X 0,Y 327.474,Z 80.562,A -85,B 0,C 180,E1 -14880.23,E2 -14880.23} C_VEL
LIN {X 0,Y 326.617,Z 76.801,A -85,B 0,C 180,E1 -14881.317,E2 -14881.317} C_VEL
LIN {X 0,Y 326.62,Z 76.8,A -85,B 0,C 180,E1 -14885.149,E2 -14885.149} C_VEL
LIN {X 0,Y 326.624,Z 76.797,A -85,B 0,C 180,E1 -14888.608,E2 -14888.608} C_VEL
LIN {X 0,Y 326.575,Z 76.806,A -85,B 0,C 180,E1 -14891.845,E2 -14891.845} C_VEL
LIN {X 0,Y 326.526,Z 76.812,A -85,B 0,C 180,E1 -14895.257,E2 -14895.257} C_VEL
LIN {X 0,Y 326.576,Z 76.804,A -85,B 0,C 180,E1 -14898.869,E2 -14898.869} C_VEL
LIN {X 0,Y 326.626,Z 76.795,A -85,B 0,C 180,E1 -14902.761,E2 -14902.761} C_VEL
LIN {X 0,Y 326.606,Z 76.799,A -85,B 0,C 180,E1 -14905.981,E2 -14905.981} C_VEL
LIN {X 0,Y 326.659,Z 76.793,A -85,B 0,C 180,E1 -14910.341,E2 -14910.341} C_VEL
LIN {X 0,Y 326.689,Z 76.789,A -85,B 0,C 180,E1 -14914.516,E2 -14914.516} C_VEL
LIN {X 0,Y 326.647,Z 76.797,A -85,B 0,C 180,E1 -14918.546,E2 -14918.546} C_VEL
LIN {X 0,Y 326.743,Z 76.782,A -85,B 0,C 180,E1 -14921.178,E2 -14921.178} C_VEL
LIN {X 0,Y 326.762,Z 76.778,A -85,B 0,C 180,E1 -14925.433,E2 -14925.433} C_VEL
LIN {X 0,Y 326.769,Z 76.779,A -85,B 0,C 180,E1 -14928.839,E2 -14928.839} C_VEL
LIN {X 0,Y 326.957,Z 76.758,A -85,B 0,C 180,E1 -14932.59,E2 -14932.59} C_VEL
LIN {X 0,Y 326.988,Z 76.753,A -85,B 0,C 180,E1 -14933.831,E2 -14933.831} C_VEL
LIN {X 0,Y 327.042,Z 76.743,A -85,B 0,C 180,E1 -14937.537,E2 -14937.537} C_VEL
LIN {X 0,Y 327.177,Z 76.732,A -85,B 0,C 180,E1 -14940,E2 -14940} C_VEL
LIN {X 0,Y 327.042,Z 76.745,A -85,B 0,C 180,E1 -14942.464,E2 -14942.464} C_VEL
LIN {X 0,Y 326.932,Z 76.758,A -85,B 0,C 180,E1 -14946.481,E2 -14946.481} C_VEL
LIN {X 0,Y 326.783,Z 76.78,A -85,B 0,C 180,E1 -14949.908,E2 -14949.908} C_VEL
LIN {X 0,Y 326.759,Z 76.782,A -85,B 0,C 180,E1 -14953.686,E2 -14953.686} C_VEL
LIN {X 0,Y 326.7,Z 76.792,A -85,B 0,C 180,E1 -14957.528,E2 -14957.528} C_VEL
LIN {X 0,Y 326.663,Z 76.79,A -85,B 0,C 180,E1 -14960.135,E2 -14960.135} C_VEL
LIN {X 0,Y 326.652,Z 76.793,A -85,B 0,C 180,E1 -14964.129,E2 -14964.129} C_VEL
LIN {X 0,Y 326.683,Z 76.791,A -85,B 0,C 180,E1 -14966.858,E2 -14966.858} C_VEL
LIN {X 0,Y 326.634,Z 76.796,A -85,B 0,C 180,E1 -14970.61,E2 -14970.61} C_VEL
LIN {X 0,Y 326.607,Z 76.798,A -85,B 0,C 180,E1 -14974.02,E2 -14974.02} C_VEL
LIN {X 0,Y 326.623,Z 76.799,A -85,B 0,C 180,E1 -14977.238,E2 -14977.238} C_VEL
LIN {X 0,Y 326.544,Z 76.809,A -85,B 0,C 180,E1 -14981.125,E2 -14981.125} C_VEL
LIN {X 0,Y 326.561,Z 76.805,A -85,B 0,C 180,E1 -14983.526,E2 -14983.526} C_VEL
LIN {X 0,Y 326.576,Z 76.804,A -85,B 0,C 180,E1 -14987.029,E2 -14987.029} C_VEL
LIN {X 0,Y 326.6,Z 76.803,A -85,B 0,C 180,E1 -14990.776,E2 -14990.776} C_VEL
LIN {X 0,Y 326.614,Z 76.802,A -85,B 0,C 180,E1 -14994.481,E2 -14994.481} C_VEL
LIN {X 0,Y 326.612,Z 76.797,A -85,B 0,C 180,E1 -14997.456,E2 -14997.456} C_VEL
LIN {X 0,Y 326.619,Z 76.798,A -85,B 0,C 180,E1 -15000.337,E2 -15000.337} C_VEL
LIN {X 0,Y 326.605,Z 76.801,A -85,B 0,C 180,E1 -15004.51,E2 -15004.51} C_VEL
LIN {X 0,Y 326.622,Z 76.798,A -85,B 0,C 180,E1 -15008.544,E2 -15008.544} C_VEL
LIN {X 0,Y 326.784,Z 76.878,A -85,B 0,C 180,E1 -15012.437,E2 -15012.437} C_VEL
LIN {X 0,Y 327.62,Z 81.092,A -85,B 0,C 180,E1 -15013.693,E2 -15013.693} C_VEL
LIN {X 0,Y 334.221,Z 100.136,A -85,B 0,C 180,E1 -15014.553,E2 -15014.553} C_VEL
LIN {X 0,Y 335.436,Z 106.552,A -85,B 0,C 180,E1 -15014.773,E2 -15014.773} C_VEL
LIN {X 0,Y 333.828,Z 187.884,A -85,B 0,C 180,E1 -15016.521,E2 -15016.521} C_VEL
LIN {X 0,Y 333.384,Z 200.461,A -85,B 0,C 180,E1 -15017.019,E2 -15017.019} C_VEL
LIN {X 0,Y 332.684,Z 212.652,A -85,B 0,C 180,E1 -15017.727,E2 -15017.727} C_VEL
LIN {X 0,Y 331.879,Z 224.938,A -85,B 0,C 180,E1 -15018.704,E2 -15018.704} C_VEL
LIN {X 0,Y 330.808,Z 236.496,A -85,B 0,C 180,E1 -15019.906,E2 -15019.906} C_VEL
LIN {X 0,Y 329.676,Z 246.896,A -85,B 0,C 180,E1 -15021.264,E2 -15021.264} C_VEL
LIN {X 0,Y 328.678,Z 255.403,A -85,B 0,C 180,E1 -15022.629,E2 -15022.629} C_VEL
LIN {X 0,Y 327.803,Z 263.239,A -85,B 0,C 180,E1 -15024.155,E2 -15024.155} C_VEL
LIN {X 0,Y 326.782,Z 270.926,A -85,B 0,C 180,E1 -15025.992,E2 -15025.992} C_VEL
LIN {X 0,Y 326.038,Z 277.973,A -85,B 0,C 180,E1 -15028.147,E2 -15028.147} C_VEL
LIN {X 0,Y 325.559,Z 282.68,A -85,B 0,C 180,E1 -15030,E2 -15030} C_VEL
LIN {X 0,Y 325.332,Z 286.285,A -85,B 0,C 180,E1 -15031.857,E2 -15031.857} C_VEL
LIN {X 0,Y 325.077,Z 288.9,A -85,B 0,C 180,E1 -15033.719,E2 -15033.719} C_VEL
LIN {X 0,Y 325.109,Z 290.881,A -85,B 0,C 180,E1 -15036.061,E2 -15036.061} C_VEL
LIN {X 0,Y 325.014,Z 291.36,A -85,B 0,C 180,E1 -15037.455,E2 -15037.455} C_VEL
LIN {X 0,Y 325.061,Z 291.026,A -85,B 0,C 180,E1 -15039.961,E2 -15039.961} C_VEL
LIN {X 0,Y 325.198,Z 290.255,A -85,B 0,C 180,E1 -15041.216,E2 -15041.216} C_VEL
LIN {X 0,Y 325.478,Z 289.046,A -85,B 0,C 180,E1 -15042.47,E2 -15042.47} C_VEL
LIN {X 0,Y 325.91,Z 287.081,A -85,B 0,C 180,E1 -15043.975,E2 -15043.975} C_VEL
LIN {X 0,Y 326.631,Z 282.856,A -85,B 0,C 180,E1 -15046.244,E2 -15046.244} C_VEL
LIN {X 0,Y 327.536,Z 278.103,A -85,B 0,C 180,E1 -15048.128,E2 -15048.128} C_VEL
LIN {X 0,Y 328.821,Z 270.937,A -85,B 0,C 180,E1 -15050.324,E2 -15050.324} C_VEL
LIN {X 0,Y 330.311,Z 263.055,A -85,B 0,C 180,E1 -15052.19,E2 -15052.19} C_VEL
LIN {X 0,Y 331.916,Z 253.748,A -85,B 0,C 180,E1 -15053.948,E2 -15053.948} C_VEL
LIN {X 0,Y 333.368,Z 243.966,A -85,B 0,C 180,E1 -15055.439,E2 -15055.439} C_VEL
LIN {X 0,Y 334.747,Z 233.889,A -85,B 0,C 180,E1 -15056.665,E2 -15056.665} C_VEL
LIN {X 0,Y 336.175,Z 222.889,A -85,B 0,C 180,E1 -15057.721,E2 -15057.721} C_VEL
LIN {X 0,Y 337.38,Z 210.673,A -85,B 0,C 180,E1 -15058.628,E2 -15058.628} C_VEL
LIN {X 0,Y 338.277,Z 198.424,A -85,B 0,C 180,E1 -15059.288,E2 -15059.288} C_VEL
LIN {X 0,Y 338.911,Z 185.149,A -85,B 0,C 180,E1 -15059.743,E2 -15059.743} C_VEL
LIN {X 0,Y 340.605,Z 115.76,A -85,B 0,C 180,E1 -15061.221,E2 -15061.221} C_VEL
LIN {X 0,Y 339.985,Z 112.738,A -85,B 0,C 180,E1 -15061.346,E2 -15061.346} C_VEL
LIN {X 0,Y 337.628,Z 109.202,A -85,B 0,C 180,E1 -15061.637,E2 -15061.637} C_VEL
LIN {X 0,Y 330.361,Z 102.195,A -85,B 0,C 180,E1 -15062.47,E2 -15062.47} C_VEL
LIN {X 0,Y 329.009,Z 99.971,A -85,B 0,C 180,E1 -15062.653,E2 -15062.653} C_VEL
LIN {X 0,Y 320.585,Z 81.879,A -85,B 0,C 180,E1 -15063.952,E2 -15063.952} C_VEL
LIN {X 0,Y 319.576,Z 77.678,A -85,B 0,C 180,E1 -15065.46,E2 -15065.46} C_VEL
LIN {X 0,Y 319.548,Z 77.681,A -85,B 0,C 180,E1 -15069.629,E2 -15069.629} C_VEL
LIN {X 0,Y 319.521,Z 77.678,A -85,B 0,C 180,E1 -15073.46,E2 -15073.46} C_VEL
LIN {X 0,Y 319.553,Z 77.68,A -85,B 0,C 180,E1 -15077.016,E2 -15077.016} C_VEL
LIN {X 0,Y 319.517,Z 77.683,A -85,B 0,C 180,E1 -15080.366,E2 -15080.366} C_VEL
LIN {X 0,Y 319.581,Z 77.671,A -85,B 0,C 180,E1 -15084.458,E2 -15084.458} C_VEL
LIN {X 0,Y 319.523,Z 77.676,A -85,B 0,C 180,E1 -15088.137,E2 -15088.137} C_VEL
LIN {X 0,Y 319.57,Z 77.673,A -85,B 0,C 180,E1 -15091.605,E2 -15091.605} C_VEL
LIN {X 0,Y 319.574,Z 77.677,A -85,B 0,C 180,E1 -15095.301,E2 -15095.301} C_VEL
LIN {X 0,Y 319.569,Z 77.67,A -85,B 0,C 180,E1 -15098.045,E2 -15098.045} C_VEL
LIN {X 0,Y 319.661,Z 77.662,A -85,B 0,C 180,E1 -15100.979,E2 -15100.979} C_VEL
LIN {X 0,Y 319.715,Z 77.659,A -85,B 0,C 180,E1 -15105.289,E2 -15105.289} C_VEL
LIN {X 0,Y 319.718,Z 77.648,A -85,B 0,C 180,E1 -15108.589,E2 -15108.589} C_VEL
LIN {X 0,Y 319.854,Z 77.636,A -85,B 0,C 180,E1 -15112.424,E2 -15112.424} C_VEL
LIN {X 0,Y 319.724,Z 77.652,A -85,B 0,C 180,E1 -15114.955,E2 -15114.955} C_VEL
LIN {X 0,Y 319.963,Z 77.628,A -85,B 0,C 180,E1 -15117.482,E2 -15117.482} C_VEL
LIN {X 0,Y 320.016,Z 77.616,A -85,B 0,C 180,E1 -15121.258,E2 -15121.258} C_VEL
LIN {X 0,Y 319.721,Z 77.65,A -85,B 0,C 180,E1 -15125.044,E2 -15125.044} C_VEL
LIN {X 0,Y 319.856,Z 77.636,A -85,B 0,C 180,E1 -15127.575,E2 -15127.575} C_VEL
LIN {X 0,Y 319.718,Z 77.647,A -85,B 0,C 180,E1 -15131.41,E2 -15131.41} C_VEL
LIN {X 0,Y 319.715,Z 77.657,A -85,B 0,C 180,E1 -15134.711,E2 -15134.711} C_VEL
LIN {X 0,Y 319.66,Z 77.663,A -85,B 0,C 180,E1 -15139.021,E2 -15139.021} C_VEL
LIN {X 0,Y 319.573,Z 77.671,A -85,B 0,C 180,E1 -15143.319,E2 -15143.319} C_VEL
LIN {X 0,Y 319.637,Z 77.664,A -85,B 0,C 180,E1 -15146.088,E2 -15146.088} C_VEL
LIN {X 0,Y 319.583,Z 77.677,A -85,B 0,C 180,E1 -15148.934,E2 -15148.934} C_VEL
LIN {X 0,Y 319.533,Z 77.68,A -85,B 0,C 180,E1 -15151.862,E2 -15151.862} C_VEL
LIN {X 0,Y 319.582,Z 77.655,A -85,B 0,C 180,E1 -15155.543,E2 -15155.543} C_VEL
LIN {X 0,Y 319.575,Z 77.665,A -85,B 0,C 180,E1 -15158.008,E2 -15158.008} C_VEL
LIN {X 0,Y 319.528,Z 77.681,A -85,B 0,C 180,E1 -15161.597,E2 -15161.597} C_VEL
LIN {X 0,Y 319.49,Z 77.686,A -85,B 0,C 180,E1 -15165.257,E2 -15165.257} C_VEL
LIN {X 0,Y 319.53,Z 77.678,A -85,B 0,C 180,E1 -15168.711,E2 -15168.711} C_VEL
LIN {X 0,Y 319.564,Z 77.676,A -85,B 0,C 180,E1 -15172.347,E2 -15172.347} C_VEL
LIN {X 0,Y 319.602,Z 77.794,A -85,B 0,C 180,E1 -15174.878,E2 -15174.878} C_VEL
LIN {X 0,Y 322.345,Z 89.049,A -85,B 0,C 180,E1 -15178.448,E2 -15178.448} C_VEL
LIN {X 0,Y 324.687,Z 99.472,A -85,B 0,C 180,E1 -15181.562,E2 -15181.562} C_VEL
LIN {X 0,Y 325.524,Z 104.684,A -85,B 0,C 180,E1 -15183.038,E2 -15183.038} C_VEL
LIN {X 0,Y 325.256,Z 106.759,A -85,B 0,C 180,E1 -15183.568,E2 -15183.568} C_VEL
LIN {X 0,Y 330.83,Z 134.653,A -85,B 0,C 180,E1 -15184.781,E2 -15184.781} C_VEL
LIN {X 0,Y 333.411,Z 151.217,A -85,B 0,C 180,E1 -15185.407,E2 -15185.407} C_VEL
LIN {X 0,Y 331.76,Z 216.239,A -85,B 0,C 180,E1 -15186.844,E2 -15186.844} C_VEL
LIN {X 0,Y 330.753,Z 230.011,A -85,B 0,C 180,E1 -15187.389,E2 -15187.389} C_VEL
LIN {X 0,Y 329.385,Z 242.894,A -85,B 0,C 180,E1 -15188.157,E2 -15188.157} C_VEL
LIN {X 0,Y 327.86,Z 254.63,A -85,B 0,C 180,E1 -15189.122,E2 -15189.122} C_VEL
LIN {X 0,Y 326.184,Z 265.954,A -85,B 0,C 180,E1 -15190.326,E2 -15190.326} C_VEL
LIN {X 0,Y 324.441,Z 276.187,A -85,B 0,C 180,E1 -15191.693,E2 -15191.693} C_VEL
LIN {X 0,Y 322.65,Z 286.368,A -85,B 0,C 180,E1 -15193.419,E2 -15193.419} C_VEL
LIN {X 0,Y 321.31,Z 294.375,A -85,B 0,C 180,E1 -15195.107,E2 -15195.107} C_VEL
LIN {X 0,Y 320.002,Z 301.627,A -85,B 0,C 180,E1 -15196.99,E2 -15196.99} C_VEL
LIN {X 0,Y 319.103,Z 306.542,A -85,B 0,C 180,E1 -15198.567,E2 -15198.567} C_VEL
LIN {X 0,Y 318.443,Z 311.34,A -85,B 0,C 180,E1 -15200.472,E2 -15200.472} C_VEL
LIN {X 0,Y 318.018,Z 315.036,A -85,B 0,C 180,E1 -15202.38,E2 -15202.38} C_VEL
LIN {X 0,Y 317.831,Z 317.743,A -85,B 0,C 180,E1 -15204.301,E2 -15204.301} C_VEL
LIN {X 0,Y 317.836,Z 319.487,A -85,B 0,C 180,E1 -15206.196,E2 -15206.196} C_VEL
LIN {X 0,Y 317.868,Z 320.43,A -85,B 0,C 180,E1 -15208.733,E2 -15208.733} C_VEL
LIN {X 0,Y 317.95,Z 320.297,A -85,B 0,C 180,E1 -15210,E2 -15210} C_VEL
LIN {X 0,Y 317.886,Z 319.733,A -85,B 0,C 180,E1 -15211.266,E2 -15211.266} C_VEL
LIN {X 0,Y 317.891,Z 317.423,A -85,B 0,C 180,E1 -15213.803,E2 -15213.803} C_VEL
LIN {X 0,Y 317.818,Z 314.591,A -85,B 0,C 180,E1 -15215.676,E2 -15215.676} C_VEL
LIN {X 0,Y 318.007,Z 310.604,A -85,B 0,C 180,E1 -15217.62,E2 -15217.62} C_VEL
LIN {X 0,Y 318.32,Z 305.524,A -85,B 0,C 180,E1 -15219.531,E2 -15219.531} C_VEL
LIN {X 0,Y 318.857,Z 299.13,A -85,B 0,C 180,E1 -15221.441,E2 -15221.441} C_VEL
LIN {X 0,Y 319.823,Z 291.124,A -85,B 0,C 180,E1 -15223.34,E2 -15223.34} C_VEL
LIN {X 0,Y 320.782,Z 282.957,A -85,B 0,C 180,E1 -15224.917,E2 -15224.917} C_VEL
LIN {X 0,Y 321.756,Z 272.968,A -85,B 0,C 180,E1 -15226.496,E2 -15226.496} C_VEL
LIN {X 0,Y 322.867,Z 263.164,A -85,B 0,C 180,E1 -15227.742,E2 -15227.742} C_VEL
LIN {X 0,Y 324.056,Z 252.554,A -85,B 0,C 180,E1 -15228.82,E2 -15228.82} C_VEL
LIN {X 0,Y 325.213,Z 239.749,A -85,B 0,C 180,E1 -15229.816,E2 -15229.816} C_VEL
LIN {X 0,Y 326.226,Z 226.933,A -85,B 0,C 180,E1 -15230.533,E2 -15230.533} C_VEL
LIN {X 0,Y 326.725,Z 214.442,A -85,B 0,C 180,E1 -15230.994,E2 -15230.994} C_VEL
LIN {X 0,Y 327.944,Z 147.87,A -85,B 0,C 180,E1 -15232.454,E2 -15232.454} C_VEL
LIN {X 0,Y 322.93,Z 110.974,A -85,B 0,C 180,E1 -15233.624,E2 -15233.624} C_VEL
LIN {X 0,Y 322.41,Z 107.175,A -85,B 0,C 180,E1 -15233.783,E2 -15233.783} C_VEL
LIN {X 0,Y 323.465,Z 97.882,A -85,B 0,C 180,E1 -15236.071,E2 -15236.071} C_VEL
LIN {X 0,Y 322.132,Z 89.46,A -85,B 0,C 180,E1 -15238.328,E2 -15238.328} C_VEL
LIN {X 0,Y 319.582,Z 77.679,A -85,B 0,C 180,E1 -15241.677,E2 -15241.677} C_VEL
LIN {X 0,Y 319.58,Z 77.68,A -85,B 0,C 180,E1 -15245.543,E2 -15245.543} C_VEL
LIN {X 0,Y 319.574,Z 77.679,A -85,B 0,C 180,E1 -15248.008,E2 -15248.008} C_VEL
LIN {X 0,Y 319.525,Z 77.686,A -85,B 0,C 180,E1 -15251.597,E2 -15251.597} C_VEL
LIN {X 0,Y 319.487,Z 77.689,A -85,B 0,C 180,E1 -15255.257,E2 -15255.257} C_VEL
LIN {X 0,Y 319.527,Z 77.681,A -85,B 0,C 180,E1 -15258.712,E2 -15258.712} C_VEL
LIN {X 0,Y 319.56,Z 77.673,A -85,B 0,C 180,E1 -15262.348,E2 -15262.348} C_VEL
LIN {X 0,Y 319.559,Z 77.681,A -85,B 0,C 180,E1 -15265.123,E2 -15265.123} C_VEL
LIN {X 0,Y 319.569,Z 77.68,A -85,B 0,C 180,E1 -15269.058,E2 -15269.058} C_VEL
LIN {X 0,Y 319.607,Z 77.672,A -85,B 0,C 180,E1 -15272.498,E2 -15272.498} C_VEL
LIN {X 0,Y 319.604,Z 77.673,A -85,B 0,C 180,E1 -15275.304,E2 -15275.304} C_VEL
LIN {X 0,Y 319.597,Z 77.672,A -85,B 0,C 180,E1 -15278.048,E2 -15278.048} C_VEL
LIN {X 0,Y 319.688,Z 77.663,A -85,B 0,C 180,E1 -15280.962,E2 -15280.962} C_VEL
LIN {X 0,Y 319.73,Z 77.655,A -85,B 0,C 180,E1 -15285.276,E2 -15285.276} C_VEL
LIN {X 0,Y 319.752,Z 77.652,A -85,B 0,C 180,E1 -15289.873,E2 -15289.873} C_VEL
LIN {X 0,Y 319.912,Z 77.637,A -85,B 0,C 180,E1 -15292.426,E2 -15292.426} C_VEL
LIN {X 0,Y 319.74,Z 77.652,A -85,B 0,C 180,E1 -15294.956,E2 -15294.956} C_VEL
LIN {X 0,Y 319.986,Z 77.622,A -85,B 0,C 180,E1 -15297.483,E2 -15297.483} C_VEL
LIN {X 0,Y 320.129,Z 77.61,A -85,B 0,C 180,E1 -15300,E2 -15300} C_VEL
LIN {X 0,Y 319.986,Z 77.623,A -85,B 0,C 180,E1 -15302.518,E2 -15302.518} C_VEL
LIN {X 0,Y 319.898,Z 77.634,A -85,B 0,C 180,E1 -15306.465,E2 -15306.465} C_VEL
LIN {X 0,Y 319.735,Z 77.656,A -85,B 0,C 180,E1 -15310.128,E2 -15310.128} C_VEL
LIN {X 0,Y 319.732,Z 77.655,A -85,B 0,C 180,E1 -15313.993,E2 -15313.993} C_VEL
LIN {X 0,Y 319.658,Z 77.665,A -85,B 0,C 180,E1 -15317.927,E2 -15317.927} C_VEL
LIN {X 0,Y 319.614,Z 77.667,A -85,B 0,C 180,E1 -15320.599,E2 -15320.599} C_VEL
LIN {X 0,Y 319.571,Z 77.678,A -85,B 0,C 180,E1 -15323.32,E2 -15323.32} C_VEL
LIN {X 0,Y 319.618,Z 77.669,A -85,B 0,C 180,E1 -15326.09,E2 -15326.09} C_VEL
LIN {X 0,Y 319.58,Z 77.677,A -85,B 0,C 180,E1 -15328.935,E2 -15328.935} C_VEL
LIN {X 0,Y 319.531,Z 77.68,A -85,B 0,C 180,E1 -15331.862,E2 -15331.862} C_VEL
LIN {X 0,Y 319.58,Z 77.675,A -85,B 0,C 180,E1 -15335.543,E2 -15335.543} C_VEL
LIN {X 0,Y 319.528,Z 77.681,A -85,B 0,C 180,E1 -15339.663,E2 -15339.663} C_VEL
LIN {X 0,Y 319.521,Z 77.682,A -85,B 0,C 180,E1 -15343.461,E2 -15343.461} C_VEL
LIN {X 0,Y 319.554,Z 77.679,A -85,B 0,C 180,E1 -15347.017,E2 -15347.017} C_VEL
LIN {X 0,Y 319.546,Z 77.683,A -85,B 0,C 180,E1 -15350.371,E2 -15350.371} C_VEL
LIN {X 0,Y 319.582,Z 77.679,A -85,B 0,C 180,E1 -15354.458,E2 -15354.458} C_VEL
LIN {X 0,Y 319.527,Z 77.684,A -85,B 0,C 180,E1 -15358.138,E2 -15358.138} C_VEL
LIN {X 0,Y 319.574,Z 77.672,A -85,B 0,C 180,E1 -15361.604,E2 -15361.604} C_VEL
LIN {X 0,Y 319.552,Z 77.678,A -85,B 0,C 180,E1 -15365.3,E2 -15365.3} C_VEL
LIN {X 0,Y 319.57,Z 77.68,A -85,B 0,C 180,E1 -15368.046,E2 -15368.046} C_VEL
LIN {X 0,Y 319.729,Z 77.672,A -85,B 0,C 180,E1 -15372.078,E2 -15372.078} C_VEL
LIN {X 0,Y 320.459,Z 81.466,A -85,B 0,C 180,E1 -15373.212,E2 -15373.212} C_VEL
LIN {X 0,Y 327.692,Z 101.895,A -85,B 0,C 180,E1 -15374.176,E2 -15374.176} C_VEL
LIN {X 0,Y 328.793,Z 108.407,A -85,B 0,C 180,E1 -15374.397,E2 -15374.397} C_VEL
LIN {X 0,Y 327.09,Z 188.873,A -85,B 0,C 180,E1 -15376.166,E2 -15376.166} C_VEL
LIN {X 0,Y 326.544,Z 201.861,A -85,B 0,C 180,E1 -15376.702,E2 -15376.702} C_VEL
LIN {X 0,Y 325.84,Z 214.32,A -85,B 0,C 180,E1 -15377.465,E2 -15377.465} C_VEL
LIN {X 0,Y 325.003,Z 226.206,A -85,B 0,C 180,E1 -15378.462,E2 -15378.462} C_VEL
LIN {X 0,Y 323.89,Z 237.589,A -85,B 0,C 180,E1 -15379.688,E2 -15379.688} C_VEL
LIN {X 0,Y 322.73,Z 247.856,A -85,B 0,C 180,E1 -15381.074,E2 -15381.074} C_VEL
LIN {X 0,Y 321.683,Z 256.259,A -85,B 0,C 180,E1 -15382.468,E2 -15382.468} C_VEL
LIN {X 0,Y 320.54,Z 265.361,A -85,B 0,C 180,E1 -15384.338,E2 -15384.338} C_VEL
LIN {X 0,Y 319.619,Z 272.688,A -85,B 0,C 180,E1 -15386.218,E2 -15386.218} C_VEL
LIN {X 0,Y 318.975,Z 278.566,A -85,B 0,C 180,E1 -15388.106,E2 -15388.106} C_VEL
LIN {X 0,Y 318.482,Z 283.215,A -85,B 0,C 180,E1 -15390,E2 -15390} C_VEL
LIN {X 0,Y 318.233,Z 286.767,A -85,B 0,C 180,E1 -15391.899,E2 -15391.899} C_VEL
LIN {X 0,Y 318,Z 289.33,A -85,B 0,C 180,E1 -15393.802,E2 -15393.802} C_VEL
LIN {X 0,Y 318.026,Z 291.162,A -85,B 0,C 180,E1 -15396.035,E2 -15396.035} C_VEL
LIN {X 0,Y 317.927,Z 291.694,A -85,B 0,C 180,E1 -15397.622,E2 -15397.622} C_VEL
LIN {X 0,Y 317.986,Z 291.312,A -85,B 0,C 180,E1 -15400.185,E2 -15400.185} C_VEL
LIN {X 0,Y 318.173,Z 290.491,A -85,B 0,C 180,E1 -15401.467,E2 -15401.467} C_VEL
LIN {X 0,Y 318.839,Z 287.621,A -85,B 0,C 180,E1 -15404.033,E2 -15404.033} C_VEL
LIN {X 0,Y 319.434,Z 284.31,A -85,B 0,C 180,E1 -15405.964,E2 -15405.964} C_VEL
LIN {X 0,Y 320.303,Z 279.899,A -85,B 0,C 180,E1 -15407.89,E2 -15407.89} C_VEL
LIN {X 0,Y 321.518,Z 273.767,A -85,B 0,C 180,E1 -15409.959,E2 -15409.959} C_VEL
LIN {X 0,Y 322.781,Z 267.139,A -85,B 0,C 180,E1 -15411.725,E2 -15411.725} C_VEL
LIN {X 0,Y 324.476,Z 258.213,A -85,B 0,C 180,E1 -15413.623,E2 -15413.623} C_VEL
LIN {X 0,Y 325.967,Z 249.19,A -85,B 0,C 180,E1 -15415.172,E2 -15415.172} C_VEL
LIN {X 0,Y 327.582,Z 238.735,A -85,B 0,C 180,E1 -15416.607,E2 -15416.607} C_VEL
LIN {X 0,Y 329.158,Z 227.27,A -85,B 0,C 180,E1 -15417.844,E2 -15417.844} C_VEL
LIN {X 0,Y 330.559,Z 215.313,A -85,B 0,C 180,E1 -15418.84,E2 -15418.84} C_VEL
LIN {X 0,Y 331.556,Z 202.893,A -85,B 0,C 180,E1 -15419.605,E2 -15419.605} C_VEL
LIN {X 0,Y 332.399,Z 189.183,A -85,B 0,C 180,E1 -15420.163,E2 -15420.163} C_VEL
LIN {X 0,Y 334.345,Z 112.915,A -85,B 0,C 180,E1 -15421.844,E2 -15421.844} C_VEL
LIN {X 0,Y 329.009,Z 99.971,A -85,B 0,C 180,E1 -15422.653,E2 -15422.653} C_VEL
LIN {X 0,Y 326.92,Z 96.967,A -85,B 0,C 180,E1 -15422.928,E2 -15422.928} C_VEL
LIN {X 0,Y 317.564,Z 89.558,A -85,B 0,C 180,E1 -15424.059,E2 -15424.059} C_VEL
LIN {X 0,Y 315.511,Z 86.557,A -85,B 0,C 180,E1 -15424.354,E2 -15424.354} C_VEL
LIN {X 0,Y 313.436,Z 82.251,A -85,B 0,C 180,E1 -15424.699,E2 -15424.699} C_VEL
LIN {X 0,Y 312.526,Z 78.56,A -85,B 0,C 180,E1 -15426.075,E2 -15426.075} C_VEL
LIN {X 0,Y 312.458,Z 78.564,A -85,B 0,C 180,E1 -15430.114,E2 -15430.114} C_VEL
LIN {X 0,Y 312.459,Z 78.55,A -85,B 0,C 180,E1 -15433.964,E2 -15433.964} C_VEL
LIN {X 0,Y 312.457,Z 78.561,A -85,B 0,C 180,E1 -15437.925,E2 -15437.925} C_VEL
LIN {X 0,Y 312.478,Z 78.559,A -85,B 0,C 180,E1 -15441.924,E2 -15441.924} C_VEL
LIN {X 0,Y 312.532,Z 78.549,A -85,B 0,C 180,E1 -15444.22,E2 -15444.22} C_VEL
LIN {X 0,Y 312.502,Z 78.556,A -85,B 0,C 180,E1 -15447.333,E2 -15447.333} C_VEL
LIN {X 0,Y 312.5,Z 78.556,A -85,B 0,C 180,E1 -15451.295,E2 -15451.295} C_VEL
LIN {X 0,Y 312.549,Z 78.552,A -85,B 0,C 180,E1 -15454.707,E2 -15454.707} C_VEL
LIN {X 0,Y 312.536,Z 78.552,A -85,B 0,C 180,E1 -15458.912,E2 -15458.912} C_VEL
LIN {X 0,Y 312.592,Z 78.538,A -85,B 0,C 180,E1 -15461.653,E2 -15461.653} C_VEL
LIN {X 0,Y 312.689,Z 78.533,A -85,B 0,C 180,E1 -15465.686,E2 -15465.686} C_VEL
LIN {X 0,Y 312.688,Z 78.531,A -85,B 0,C 180,E1 -15469.641,E2 -15469.641} C_VEL
LIN {X 0,Y 312.798,Z 78.517,A -85,B 0,C 180,E1 -15472.252,E2 -15472.252} C_VEL
LIN {X 0,Y 312.694,Z 78.526,A -85,B 0,C 180,E1 -15474.842,E2 -15474.842} C_VEL
LIN {X 0,Y 312.971,Z 78.49,A -85,B 0,C 180,E1 -15478.713,E2 -15478.713} C_VEL
LIN {X 0,Y 312.983,Z 78.492,A -85,B 0,C 180,E1 -15481.286,E2 -15481.286} C_VEL
LIN {X 0,Y 312.844,Z 78.503,A -85,B 0,C 180,E1 -15486.449,E2 -15486.449} C_VEL
LIN {X 0,Y 312.754,Z 78.525,A -85,B 0,C 180,E1 -15489.05,E2 -15489.05} C_VEL
LIN {X 0,Y 312.637,Z 78.533,A -85,B 0,C 180,E1 -15492.991,E2 -15492.991} C_VEL
LIN {X 0,Y 312.624,Z 78.538,A -85,B 0,C 180,E1 -15495.65,E2 -15495.65} C_VEL
LIN {X 0,Y 312.58,Z 78.549,A -85,B 0,C 180,E1 -15499.71,E2 -15499.71} C_VEL
LIN {X 0,Y 312.549,Z 78.542,A -85,B 0,C 180,E1 -15502.789,E2 -15502.789} C_VEL
LIN {X 0,Y 312.605,Z 78.54,A -85,B 0,C 180,E1 -15505.935,E2 -15505.935} C_VEL
LIN {X 0,Y 312.541,Z 78.551,A -85,B 0,C 180,E1 -15509.65,E2 -15509.65} C_VEL
LIN {X 0,Y 312.522,Z 78.553,A -85,B 0,C 180,E1 -15513.688,E2 -15513.688} C_VEL
LIN {X 0,Y 312.528,Z 78.533,A -85,B 0,C 180,E1 -15517.385,E2 -15517.385} C_VEL
LIN {X 0,Y 312.492,Z 78.557,A -85,B 0,C 180,E1 -15520.709,E2 -15520.709} C_VEL
LIN {X 0,Y 312.454,Z 78.565,A -85,B 0,C 180,E1 -15524.209,E2 -15524.209} C_VEL
LIN {X 0,Y 312.486,Z 78.557,A -85,B 0,C 180,E1 -15527.918,E2 -15527.918} C_VEL
LIN {X 0,Y 312.508,Z 78.555,A -85,B 0,C 180,E1 -15531.917,E2 -15531.917} C_VEL
LIN {X 0,Y 312.553,Z 78.605,A -85,B 0,C 180,E1 -15534.223,E2 -15534.223} C_VEL
LIN {X 0,Y 315.307,Z 89.784,A -85,B 0,C 180,E1 -15537.887,E2 -15537.887} C_VEL
LIN {X 0,Y 317.728,Z 100.627,A -85,B 0,C 180,E1 -15541.218,E2 -15541.218} C_VEL
LIN {X 0,Y 318.672,Z 106.636,A -85,B 0,C 180,E1 -15542.915,E2 -15542.915} C_VEL
LIN {X 0,Y 323.75,Z 131.589,A -85,B 0,C 180,E1 -15544.045,E2 -15544.045} C_VEL
LIN {X 0,Y 327.112,Z 152.156,A -85,B 0,C 180,E1 -15544.865,E2 -15544.865} C_VEL
LIN {X 0,Y 325.415,Z 215.452,A -85,B 0,C 180,E1 -15546.281,E2 -15546.281} C_VEL
LIN {X 0,Y 324.457,Z 228.617,A -85,B 0,C 180,E1 -15546.799,E2 -15546.799} C_VEL
LIN {X 0,Y 323.08,Z 241.287,A -85,B 0,C 180,E1 -15547.539,E2 -15547.539} C_VEL
LIN {X 0,Y 321.476,Z 253.355,A -85,B 0,C 180,E1 -15548.519,E2 -15548.519} C_VEL
LIN {X 0,Y 319.737,Z 264.85,A -85,B 0,C 180,E1 -15549.745,E2 -15549.745} C_VEL
LIN {X 0,Y 317.885,Z 275.225,A -85,B 0,C 180,E1 -15551.135,E2 -15551.135} C_VEL
LIN {X 0,Y 316.309,Z 283.721,A -85,B 0,C 180,E1 -15552.545,E2 -15552.545} C_VEL
LIN {X 0,Y 314.639,Z 292.958,A -85,B 0,C 180,E1 -15554.452,E2 -15554.452} C_VEL
LIN {X 0,Y 313.266,Z 300.4,A -85,B 0,C 180,E1 -15556.375,E2 -15556.375} C_VEL
LIN {X 0,Y 312.105,Z 306.395,A -85,B 0,C 180,E1 -15558.307,E2 -15558.307} C_VEL
LIN {X 0,Y 311.399,Z 311.155,A -85,B 0,C 180,E1 -15560.254,E2 -15560.254} C_VEL
LIN {X 0,Y 310.97,Z 314.816,A -85,B 0,C 180,E1 -15562.206,E2 -15562.206} C_VEL
LIN {X 0,Y 310.727,Z 317.727,A -85,B 0,C 180,E1 -15564.378,E2 -15564.378} C_VEL
LIN {X 0,Y 310.743,Z 319.204,A -85,B 0,C 180,E1 -15566.109,E2 -15566.109} C_VEL
LIN {X 0,Y 310.775,Z 320.116,A -85,B 0,C 180,E1 -15568.704,E2 -15568.704} C_VEL
LIN {X 0,Y 310.857,Z 319.953,A -85,B 0,C 180,E1 -15570,E2 -15570} C_VEL
LIN {X 0,Y 310.792,Z 319.374,A -85,B 0,C 180,E1 -15571.295,E2 -15571.295} C_VEL
LIN {X 0,Y 310.769,Z 318.402,A -85,B 0,C 180,E1 -15572.592,E2 -15572.592} C_VEL
LIN {X 0,Y 310.793,Z 317.032,A -85,B 0,C 180,E1 -15573.89,E2 -15573.89} C_VEL
LIN {X 0,Y 310.723,Z 314.486,A -85,B 0,C 180,E1 -15575.614,E2 -15575.614} C_VEL
LIN {X 0,Y 310.955,Z 310.146,A -85,B 0,C 180,E1 -15577.793,E2 -15577.793} C_VEL
LIN {X 0,Y 311.369,Z 304.034,A -85,B 0,C 180,E1 -15580.074,E2 -15580.074} C_VEL
LIN {X 0,Y 312.004,Z 297.328,A -85,B 0,C 180,E1 -15582.026,E2 -15582.026} C_VEL
LIN {X 0,Y 312.979,Z 289.003,A -85,B 0,C 180,E1 -15583.968,E2 -15583.968} C_VEL
LIN {X 0,Y 314.081,Z 280.474,A -85,B 0,C 180,E1 -15585.576,E2 -15585.576} C_VEL
LIN {X 0,Y 315.121,Z 269.889,A -85,B 0,C 180,E1 -15587.188,E2 -15587.188} C_VEL
LIN {X 0,Y 316.463,Z 259.45,A -85,B 0,C 180,E1 -15588.449,E2 -15588.449} C_VEL
LIN {X 0,Y 317.69,Z 247.981,A -85,B 0,C 180,E1 -15589.548,E2 -15589.548} C_VEL
LIN {X 0,Y 318.746,Z 236.152,A -85,B 0,C 180,E1 -15590.404,E2 -15590.404} C_VEL
LIN {X 0,Y 319.637,Z 223.41,A -85,B 0,C 180,E1 -15591.06,E2 -15591.06} C_VEL
LIN {X 0,Y 320.167,Z 210.277,A -85,B 0,C 180,E1 -15591.488,E2 -15591.488} C_VEL
LIN {X 0,Y 321.272,Z 148.718,A -85,B 0,C 180,E1 -15592.853,E2 -15592.853} C_VEL
LIN {X 0,Y 316.384,Z 112.429,A -85,B 0,C 180,E1 -15594.034,E2 -15594.034} C_VEL
LIN {X 0,Y 315.562,Z 106.99,A -85,B 0,C 180,E1 -15594.225,E2 -15594.225} C_VEL
LIN {X 0,Y 316.472,Z 98.503,A -85,B 0,C 180,E1 -15596.368,E2 -15596.368} C_VEL
LIN {X 0,Y 315.079,Z 90.199,A -85,B 0,C 180,E1 -15598.657,E2 -15598.657} C_VEL
LIN {X 0,Y 312.527,Z 78.559,A -85,B 0,C 180,E1 -15602.048,E2 -15602.048} C_VEL
LIN {X 0,Y 312.536,Z 78.558,A -85,B 0,C 180,E1 -15605.95,E2 -15605.95} C_VEL
LIN {X 0,Y 312.508,Z 78.557,A -85,B 0,C 180,E1 -15609.027,E2 -15609.027} C_VEL
LIN {X 0,Y 312.489,Z 78.558,A -85,B 0,C 180,E1 -15612.431,E2 -15612.431} C_VEL
LIN {X 0,Y 312.457,Z 78.563,A -85,B 0,C 180,E1 -15616.035,E2 -15616.035} C_VEL
LIN {X 0,Y 312.503,Z 78.553,A -85,B 0,C 180,E1 -15619.874,E2 -15619.874} C_VEL
LIN {X 0,Y 312.534,Z 78.551,A -85,B 0,C 180,E1 -15624.05,E2 -15624.05} C_VEL
LIN {X 0,Y 312.503,Z 78.559,A -85,B 0,C 180,E1 -15627.334,E2 -15627.334} C_VEL
LIN {X 0,Y 312.551,Z 78.552,A -85,B 0,C 180,E1 -15631.276,E2 -15631.276} C_VEL
LIN {X 0,Y 312.584,Z 78.547,A -85,B 0,C 180,E1 -15634.711,E2 -15634.711} C_VEL
LIN {X 0,Y 312.586,Z 78.545,A -85,B 0,C 180,E1 -15637.529,E2 -15637.529} C_VEL
LIN {X 0,Y 312.637,Z 78.538,A -85,B 0,C 180,E1 -15641.657,E2 -15641.657} C_VEL
LIN {X 0,Y 312.693,Z 78.531,A -85,B 0,C 180,E1 -15645.686,E2 -15645.686} C_VEL
LIN {X 0,Y 312.697,Z 78.53,A -85,B 0,C 180,E1 -15649.642,E2 -15649.642} C_VEL
LIN {X 0,Y 312.853,Z 78.517,A -85,B 0,C 180,E1 -15652.254,E2 -15652.254} C_VEL
LIN {X 0,Y 312.71,Z 78.528,A -85,B 0,C 180,E1 -15654.843,E2 -15654.843} C_VEL
LIN {X 0,Y 312.985,Z 78.496,A -85,B 0,C 180,E1 -15658.714,E2 -15658.714} C_VEL
LIN {X 0,Y 312.986,Z 78.495,A -85,B 0,C 180,E1 -15661.287,E2 -15661.287} C_VEL
LIN {X 0,Y 312.703,Z 78.526,A -85,B 0,C 180,E1 -15665.158,E2 -15665.158} C_VEL
LIN {X 0,Y 312.818,Z 78.519,A -85,B 0,C 180,E1 -15667.747,E2 -15667.747} C_VEL
LIN {X 0,Y 312.663,Z 78.537,A -85,B 0,C 180,E1 -15671.672,E2 -15671.672} C_VEL
LIN {X 0,Y 312.7,Z 78.529,A -85,B 0,C 180,E1 -15674.888,E2 -15674.888} C_VEL
LIN {X 0,Y 312.63,Z 78.542,A -85,B 0,C 180,E1 -15679.237,E2 -15679.237} C_VEL
LIN {X 0,Y 312.546,Z 78.548,A -85,B 0,C 180,E1 -15682.79,E2 -15682.79} C_VEL
LIN {X 0,Y 312.597,Z 78.544,A -85,B 0,C 180,E1 -15685.934,E2 -15685.934} C_VEL
LIN {X 0,Y 312.539,Z 78.552,A -85,B 0,C 180,E1 -15689.651,E2 -15689.651} C_VEL
LIN {X 0,Y 312.52,Z 78.554,A -85,B 0,C 180,E1 -15693.689,E2 -15693.689} C_VEL
LIN {X 0,Y 312.514,Z 78.555,A -85,B 0,C 180,E1 -15697.387,E2 -15697.387} C_VEL
LIN {X 0,Y 312.441,Z 78.568,A -85,B 0,C 180,E1 -15700.718,E2 -15700.718} C_VEL
LIN {X 0,Y 312.452,Z 78.564,A -85,B 0,C 180,E1 -15704.21,E2 -15704.21} C_VEL
LIN {X 0,Y 312.468,Z 78.56,A -85,B 0,C 180,E1 -15707.923,E2 -15707.923} C_VEL
LIN {X 0,Y 312.496,Z 78.558,A -85,B 0,C 180,E1 -15710.971,E2 -15710.971} C_VEL
LIN {X 0,Y 312.533,Z 78.556,A -85,B 0,C 180,E1 -15714.221,E2 -15714.221} C_VEL
LIN {X 0,Y 312.504,Z 78.554,A -85,B 0,C 180,E1 -15717.334,E2 -15717.334} C_VEL
LIN {X 0,Y 312.509,Z 78.55,A -85,B 0,C 180,E1 -15721.292,E2 -15721.292} C_VEL
LIN {X 0,Y 312.527,Z 78.554,A -85,B 0,C 180,E1 -15724.706,E2 -15724.706} C_VEL
LIN {X 0,Y 312.564,Z 78.551,A -85,B 0,C 180,E1 -15727.528,E2 -15727.528} C_VEL
LIN {X 0,Y 312.705,Z 78.611,A -85,B 0,C 180,E1 -15731.746,E2 -15731.746} C_VEL
LIN {X 0,Y 313.328,Z 81.732,A -85,B 0,C 180,E1 -15732.708,E2 -15732.708} C_VEL
LIN {X 0,Y 321.193,Z 103.87,A -85,B 0,C 180,E1 -15733.791,E2 -15733.791} C_VEL
LIN {X 0,Y 322.145,Z 108.656,A -85,B 0,C 180,E1 -15733.967,E2 -15733.967} C_VEL
LIN {X 0,Y 320.395,Z 188.637,A -85,B 0,C 180,E1 -15735.753,E2 -15735.753} C_VEL
LIN {X 0,Y 319.84,Z 201.728,A -85,B 0,C 180,E1 -15736.297,E2 -15736.297} C_VEL
LIN {X 0,Y 319.111,Z 213.754,A -85,B 0,C 180,E1 -15737.035,E2 -15737.035} C_VEL
LIN {X 0,Y 318.257,Z 225.901,A -85,B 0,C 180,E1 -15738.052,E2 -15738.052} C_VEL
LIN {X 0,Y 317.087,Z 237.402,A -85,B 0,C 180,E1 -15739.303,E2 -15739.303} C_VEL
LIN {X 0,Y 315.883,Z 247.756,A -85,B 0,C 180,E1 -15740.718,E2 -15740.718} C_VEL
LIN {X 0,Y 314.689,Z 257.091,A -85,B 0,C 180,E1 -15742.3,E2 -15742.3} C_VEL
LIN {X 0,Y 313.501,Z 266.087,A -85,B 0,C 180,E1 -15744.211,E2 -15744.211} C_VEL
LIN {X 0,Y 312.572,Z 273.342,A -85,B 0,C 180,E1 -15746.133,E2 -15746.133} C_VEL
LIN {X 0,Y 311.914,Z 279.156,A -85,B 0,C 180,E1 -15748.064,E2 -15748.064} C_VEL
LIN {X 0,Y 311.407,Z 283.749,A -85,B 0,C 180,E1 -15750,E2 -15750} C_VEL
LIN {X 0,Y 311.258,Z 286.185,A -85,B 0,C 180,E1 -15751.294,E2 -15751.294} C_VEL
LIN {X 0,Y 310.978,Z 288.182,A -85,B 0,C 180,E1 -15752.591,E2 -15752.591} C_VEL
LIN {X 0,Y 310.926,Z 289.76,A -85,B 0,C 180,E1 -15753.889,E2 -15753.889} C_VEL
LIN {X 0,Y 310.94,Z 291.438,A -85,B 0,C 180,E1 -15756.002,E2 -15756.002} C_VEL
LIN {X 0,Y 310.842,Z 292.029,A -85,B 0,C 180,E1 -15757.797,E2 -15757.797} C_VEL
LIN {X 0,Y 310.849,Z 292.006,A -85,B 0,C 180,E1 -15759.107,E2 -15759.107} C_VEL
LIN {X 0,Y 310.92,Z 291.588,A -85,B 0,C 180,E1 -15760.419,E2 -15760.419} C_VEL
LIN {X 0,Y 311.156,Z 290.728,A -85,B 0,C 180,E1 -15761.729,E2 -15761.729} C_VEL
LIN {X 0,Y 311.851,Z 287.809,A -85,B 0,C 180,E1 -15764.354,E2 -15764.354} C_VEL
LIN {X 0,Y 312.511,Z 284.445,A -85,B 0,C 180,E1 -15766.327,E2 -15766.327} C_VEL
LIN {X 0,Y 313.443,Z 279.976,A -85,B 0,C 180,E1 -15768.295,E2 -15768.295} C_VEL
LIN {X 0,Y 314.83,Z 273.146,A -85,B 0,C 180,E1 -15770.585,E2 -15770.585} C_VEL
LIN {X 0,Y 316.38,Z 265.687,A -85,B 0,C 180,E1 -15772.532,E2 -15772.532} C_VEL
LIN {X 0,Y 317.874,Z 258.043,A -85,B 0,C 180,E1 -15774.144,E2 -15774.144} C_VEL
LIN {X 0,Y 319.346,Z 249.376,A -85,B 0,C 180,E1 -15775.651,E2 -15775.651} C_VEL
LIN {X 0,Y 320.944,Z 239.583,A -85,B 0,C 180,E1 -15777.026,E2 -15777.026} C_VEL
LIN {X 0,Y 322.599,Z 228.239,A -85,B 0,C 180,E1 -15778.284,E2 -15778.284} C_VEL
LIN {X 0,Y 324.059,Z 216.455,A -85,B 0,C 180,E1 -15779.297,E2 -15779.297} C_VEL
LIN {X 0,Y 325.042,Z 204.856,A -85,B 0,C 180,E1 -15780.056,E2 -15780.056} C_VEL
LIN {X 0,Y 325.9,Z 192,A -85,B 0,C 180,E1 -15780.625,E2 -15780.625} C_VEL
LIN {X 0,Y 326.528,Z 173.136,A -85,B 0,C 180,E1 -15781.102,E2 -15781.102} C_VEL
LIN {X 0,Y 328.041,Z 114.69,A -85,B 0,C 180,E1 -15782.385,E2 -15782.385} C_VEL
LIN {X 0,Y 321.223,Z 98.625,A -85,B 0,C 180,E1 -15783.451,E2 -15783.451} C_VEL
LIN {X 0,Y 315.511,Z 86.557,A -85,B 0,C 180,E1 -15784.354,E2 -15784.354} C_VEL
LIN {X 0,Y 313.883,Z 84.121,A -85,B 0,C 180,E1 -15784.641,E2 -15784.641} C_VEL
LIN {X 0,Y 311.055,Z 81.92,A -85,B 0,C 180,E1 -15785.215,E2 -15785.215} C_VEL
LIN {X 0,Y 307.94,Z 80.415,A -85,B 0,C 180,E1 -15786.035,E2 -15786.035} C_VEL
LIN {X 0,Y 305.961,Z 79.622,A -85,B 0,C 180,E1 -15786.874,E2 -15786.874} C_VEL
LIN {X 0,Y 305.438,Z 79.432,A -85,B 0,C 180,E1 -15787.526,E2 -15787.526} C_VEL
LIN {X 0,Y 305.414,Z 79.441,A -85,B 0,C 180,E1 -15791.862,E2 -15791.862} C_VEL
LIN {X 0,Y 305.401,Z 79.428,A -85,B 0,C 180,E1 -15795.511,E2 -15795.511} C_VEL
LIN {X 0,Y 305.414,Z 79.437,A -85,B 0,C 180,E1 -15798.138,E2 -15798.138} C_VEL
LIN {X 0,Y 305.444,Z 79.434,A -85,B 0,C 180,E1 -15801.592,E2 -15801.592} C_VEL
LIN {X 0,Y 305.464,Z 79.429,A -85,B 0,C 180,E1 -15804.886,E2 -15804.886} C_VEL
LIN {X 0,Y 305.442,Z 79.429,A -85,B 0,C 180,E1 -15808.359,E2 -15808.359} C_VEL
LIN {X 0,Y 305.466,Z 79.434,A -85,B 0,C 180,E1 -15811.108,E2 -15811.108} C_VEL
LIN {X 0,Y 305.5,Z 79.428,A -85,B 0,C 180,E1 -15814.081,E2 -15814.081} C_VEL
LIN {X 0,Y 305.477,Z 79.424,A -85,B 0,C 180,E1 -15816.976,E2 -15816.976} C_VEL
LIN {X 0,Y 305.552,Z 79.417,A -85,B 0,C 180,E1 -15821.215,E2 -15821.215} C_VEL
LIN {X 0,Y 305.63,Z 79.414,A -85,B 0,C 180,E1 -15825.348,E2 -15825.348} C_VEL
LIN {X 0,Y 305.627,Z 79.41,A -85,B 0,C 180,E1 -15829.399,E2 -15829.399} C_VEL
LIN {X 0,Y 305.748,Z 79.397,A -85,B 0,C 180,E1 -15832.072,E2 -15832.072} C_VEL
LIN {X 0,Y 305.664,Z 79.4,A -85,B 0,C 180,E1 -15834.723,E2 -15834.723} C_VEL
LIN {X 0,Y 305.939,Z 79.366,A -85,B 0,C 180,E1 -15838.683,E2 -15838.683} C_VEL
LIN {X 0,Y 305.95,Z 79.368,A -85,B 0,C 180,E1 -15841.316,E2 -15841.316} C_VEL
LIN {X 0,Y 305.789,Z 79.382,A -85,B 0,C 180,E1 -15846.599,E2 -15846.599} C_VEL
LIN {X 0,Y 305.697,Z 79.405,A -85,B 0,C 180,E1 -15849.261,E2 -15849.261} C_VEL
LIN {X 0,Y 305.59,Z 79.412,A -85,B 0,C 180,E1 -15853.296,E2 -15853.296} C_VEL
LIN {X 0,Y 305.554,Z 79.415,A -85,B 0,C 180,E1 -15856.022,E2 -15856.022} C_VEL
LIN {X 0,Y 305.564,Z 79.422,A -85,B 0,C 180,E1 -15859.436,E2 -15859.436} C_VEL
LIN {X 0,Y 305.493,Z 79.422,A -85,B 0,C 180,E1 -15863.041,E2 -15863.041} C_VEL
LIN {X 0,Y 305.549,Z 79.418,A -85,B 0,C 180,E1 -15866.226,E2 -15866.226} C_VEL
LIN {X 0,Y 305.491,Z 79.434,A -85,B 0,C 180,E1 -15869.047,E2 -15869.047} C_VEL
LIN {X 0,Y 305.444,Z 79.435,A -85,B 0,C 180,E1 -15871.952,E2 -15871.952} C_VEL
LIN {X 0,Y 305.464,Z 79.417,A -85,B 0,C 180,E1 -15875.113,E2 -15875.113} C_VEL
LIN {X 0,Y 305.469,Z 79.427,A -85,B 0,C 180,E1 -15878.532,E2 -15878.532} C_VEL
LIN {X 0,Y 305.457,Z 79.438,A -85,B 0,C 180,E1 -15882.585,E2 -15882.585} C_VEL
LIN {X 0,Y 305.427,Z 79.435,A -85,B 0,C 180,E1 -15886.345,E2 -15886.345} C_VEL
LIN {X 0,Y 305.46,Z 79.432,A -85,B 0,C 180,E1 -15889.892,E2 -15889.892} C_VEL
LIN {X 0,Y 305.496,Z 79.551,A -85,B 0,C 180,E1 -15893.572,E2 -15893.572} C_VEL
LIN {X 0,Y 308.131,Z 90.027,A -85,B 0,C 180,E1 -15897.134,E2 -15897.134} C_VEL
LIN {X 0,Y 310.801,Z 101.954,A -85,B 0,C 180,E1 -15900.91,E2 -15900.91} C_VEL
LIN {X 0,Y 311.646,Z 106.305,A -85,B 0,C 180,E1 -15902.169,E2 -15902.169} C_VEL
LIN {X 0,Y 313.295,Z 111.533,A -85,B 0,C 180,E1 -15902.481,E2 -15902.481} C_VEL
LIN {X 0,Y 318.318,Z 137.082,A -85,B 0,C 180,E1 -15903.652,E2 -15903.652} C_VEL
LIN {X 0,Y 320.815,Z 152.821,A -85,B 0,C 180,E1 -15904.291,E2 -15904.291} C_VEL
LIN {X 0,Y 319.037,Z 215.799,A -85,B 0,C 180,E1 -15905.733,E2 -15905.733} C_VEL
LIN {X 0,Y 317.968,Z 229.502,A -85,B 0,C 180,E1 -15906.297,E2 -15906.297} C_VEL
LIN {X 0,Y 316.548,Z 241.833,A -85,B 0,C 180,E1 -15907.05,E2 -15907.05} C_VEL
LIN {X 0,Y 314.909,Z 253.659,A -85,B 0,C 180,E1 -15908.048,E2 -15908.048} C_VEL
LIN {X 0,Y 313.105,Z 265.04,A -85,B 0,C 180,E1 -15909.296,E2 -15909.296} C_VEL
LIN {X 0,Y 311.164,Z 275.325,A -85,B 0,C 180,E1 -15910.711,E2 -15910.711} C_VEL
LIN {X 0,Y 309.193,Z 285.393,A -85,B 0,C 180,E1 -15912.471,E2 -15912.471} C_VEL
LIN {X 0,Y 307.519,Z 294.261,A -85,B 0,C 180,E1 -15914.423,E2 -15914.423} C_VEL
LIN {X 0,Y 306.14,Z 301.408,A -85,B 0,C 180,E1 -15916.39,E2 -15916.39} C_VEL
LIN {X 0,Y 305.112,Z 306.25,A -85,B 0,C 180,E1 -15918.035,E2 -15918.035} C_VEL
LIN {X 0,Y 304.373,Z 310.972,A -85,B 0,C 180,E1 -15920.027,E2 -15920.027} C_VEL
LIN {X 0,Y 303.916,Z 314.597,A -85,B 0,C 180,E1 -15922.024,E2 -15922.024} C_VEL
LIN {X 0,Y 303.625,Z 317.693,A -85,B 0,C 180,E1 -15924.455,E2 -15924.455} C_VEL
LIN {X 0,Y 303.652,Z 318.921,A -85,B 0,C 180,E1 -15926.018,E2 -15926.018} C_VEL
LIN {X 0,Y 303.655,Z 319.556,A -85,B 0,C 180,E1 -15927.346,E2 -15927.346} C_VEL
LIN {X 0,Y 303.684,Z 319.799,A -85,B 0,C 180,E1 -15928.674,E2 -15928.674} C_VEL
LIN {X 0,Y 303.764,Z 319.609,A -85,B 0,C 180,E1 -15930,E2 -15930} C_VEL
LIN {X 0,Y 303.702,Z 319.014,A -85,B 0,C 180,E1 -15931.326,E2 -15931.326} C_VEL
LIN {X 0,Y 303.69,Z 318.028,A -85,B 0,C 180,E1 -15932.652,E2 -15932.652} C_VEL
LIN {X 0,Y 303.699,Z 316.636,A -85,B 0,C 180,E1 -15933.981,E2 -15933.981} C_VEL
